Omron CX-Programmer project NewProject (CX-Programmer 9.75)

# PLC NewPLC1: CP1L M

## Global symbols (name address type ; comment)
0.00 BOOL  ; I_CYL-
0.01 BOOL  ; I_CYL+
0.02 BOOL  ; I_D-RED
0.03 BOOL  ; I_D-SILVER
0.04 BOOL  ; I_D-BLACK
0.05 BOOL  ; I_D-ENABLE V
0.06 BOOL  ; I_D-ENABLE H
0.07 BOOL  ; I_IP/FI
0.08 BOOL  ; I_PB START
0.09 BOOL  ; I_PB STOP
0.10 BOOL  ; I_SELECTOR
0.11 BOOL  ; I_RESET
100.00 BOOL  ; O_CYLINDER
100.01 BOOL  ; O_GRIPPER
100.02 BOOL  ; O_BIT 1
100.03 BOOL  ; O_BIT 2
100.04 BOOL  ; O_BIT 3
100.05 BOOL  ; O_ENABLE VERTICAL
100.06 BOOL  ; O_ENABLE HORIZONTAL
100.07 BOOL  ; O_START LAMP
101.00 BOOL  ; O_RESET LAMP
101.01 BOOL  ; O_Q1 LAMP
101.02 BOOL  ; O_Q2 LAMP
101.03 BOOL  ; O_Q4 LAMP
10.00 BOOL  ; O_IM_CYLINDER
10.01 BOOL  ; O_IM_GRIPPER
10.02 BOOL  ; O_IM_BIT 1
10.03 BOOL  ; O_IM_BIT 2
10.04 BOOL  ; O_IM_BIT 3
10.05 BOOL  ; O_IM_ENABLE VERTICAL
10.06 BOOL  ; O_IM_ENABLE HORIZONTAL
10.07 BOOL  ; O_IM_START LAMP
11.00 BOOL  ; O_IM_RESET LAMP
11.01 BOOL  ; O_IM_Q1 LAMP
11.02 BOOL  ; O_IM_Q2 LAMP
11.03 BOOL  ; O_IM_Q4 LAMP
11.04 BOOL  ; O_IM_PROGRAM BLINK
20.01 BOOL  ; SEQ1
20.02 BOOL  ; SEQ2
20.03 BOOL  ; SEQ3
20.04 BOOL  ; SEQ4
20.05 BOOL  ; SEQ5
20.06 BOOL  ; SEQ6
20.07 BOOL  ; SEQ7
20.08 BOOL  ; SEQ8
20.09 BOOL  ; SEQ9
20.10 BOOL  ; SEQ10
20.11 BOOL  ; SEQ11
20.12 BOOL  ; SEQ12
20.13 BOOL  ; SEQ13
20.14 BOOL  ; SEQ14
20.15 BOOL  ; SEQ15
21.06 BOOL  ; SEQ16
21.07 BOOL  ; SEQ17
21.08 BOOL  ; SEQ18
21.09 BOOL  ; SEQ19
22.00 BOOL  ; SEQ20
22.01 BOOL  ; SEQ21
22.02 BOOL  ; SEQ22
22.03 BOOL  ; SEQ23
30.01 BOOL  ; P_CAL1
30.02 BOOL  ; P_CAL2
30.03 BOOL  ; P_CAL3
30.04 BOOL  ; P_CAL4
30.05 BOOL  ; P_CAL5
30.06 BOOL  ; P_CAL6
30.07 BOOL  ; WP_RED
30.08 BOOL  ; WP_SILVER
30.09 BOOL  ; WP_BLACK
30.10 BOOL  ; CALIBRATION ON
30.11 BOOL  ; P_S_STOP-FUNCTION
30.12 BOOL  ; P_EMG-ACTIVE
30.13 BOOL  ; P_CAL-LAMP
30.14 BOOL  ; P_N_Send/5s
30.15 BOOL  ; P_ST_OFF LAMP
31.00 BOOL  ; P_EMERGENCY-1
31.01 BOOL  ; P_EMERGENCY-2
31.02 BOOL  ; P_EMERGENCY-3
31.03 BOOL  ; P_EMERGENCY-4
31.04 BOOL  ; DEACT WHEN RESET ON
32.00 BOOL  ; P_RST-SEQ1
32.01 BOOL  ; P_RST-SEQ2
32.02 BOOL  ; P_RST-SEQ3
32.03 BOOL  ; P_RST-SEQ4
32.04 BOOL  ; P_RST-SEQ5
32.05 BOOL  ; P_RST-SEQ6
32.06 BOOL  ; P_RST-SEQ7
32.07 BOOL  ; P_RST-SEQ8
32.08 BOOL  ; P_RST-SEQ9
32.09 BOOL  ; MANUAL RESET
32.10 BOOL  ; PB RESET HELPER
40.01 BOOL  ; SEQ-1
40.02 BOOL  ; SEQ-2
40.03 BOOL  ; SEQ-3
40.04 BOOL  ; SEQ-4
40.05 BOOL  ; SEQ-5
40.06 BOOL  ; SEQ-6
40.07 BOOL  ; SEQ-7
40.08 BOOL  ; SEQ-8
40.09 BOOL  ; SEQ-9
40.10 BOOL  ; SEQ-10
40.11 BOOL  ; SEQ-11
40.12 BOOL  ; SEQ-12
40.13 BOOL  ; SEQ-13
40.14 BOOL  ; SEQ-14
40.15 BOOL  ; SEQ-15
70.00 BOOL  ; HAPUS
70.01 BOOL  ; UBAH HMI UNTUK NON AKTIFKAN SELFHOLDING
70.02 BOOL  ; EMG PROTOTYPE
70.03 BOOL  ; TRIAL
70.04 BOOL  ; TRIAL-2
80.00 BOOL  ; CALIBRATION V
80.01 BOOL  ; LT1
80.02 BOOL  ; LT2
80.03 BOOL  ; LT3
80.04 BOOL  ; HOME
80.05 BOOL  ; PICKUP
80.07 BOOL  ; S_MOVE-V
80.08 BOOL  ; HELPER SEQ-V
80.09 BOOL  ; HELPER SEQ-V
80.10 BOOL  ; HELPER SEQ-V3
81.01 BOOL  ; POSITION 1
81.02 BOOL  ; POSITION 2
81.03 BOOL  ; POSITION 3
81.04 BOOL  ; POSITION 4
81.05 BOOL  ; POSITION 5
81.06 BOOL  ; POSITION 6
81.07 BOOL  ; HOME
81.08 BOOL  ; CALIBRATION
81.09 BOOL  ; S_MOVE-H
81.10 BOOL  ; HELPER SEQ-H
81.11 BOOL  ; HELPER SEQ-H-2
81.12 BOOL  ; HELPER SEQ-H-3
81.13 BOOL  ; HELPER H
85.00 BOOL  ; PL_LA_RED-L1
85.01 BOOL  ; PL_LA_RED-L2
85.02 BOOL  ; PL_LA_RED-L3
85.03 BOOL  ; PL_LA_SILVER-L1
85.04 BOOL  ; PL_LA_SILVER-L2
85.05 BOOL  ; PL_LA_SILVER-L3
85.06 BOOL  ; PL_LA_BLACK-L1
85.07 BOOL  ; PL_LA_BLACK-L2
85.08 BOOL  ; PL_LA_BLACK-L3
86.01 BOOL  ; PP_L3_P1
86.02 BOOL  ; PP_L3_P2
86.03 BOOL  ; PP_L3_P3
86.04 BOOL  ; PP_L3_P4
86.05 BOOL  ; PP_L3_P5
86.06 BOOL  ; PP_L3_P6
87.01 BOOL  ; PP_L2_P1
87.02 BOOL  ; PP_L2_P2
87.03 BOOL  ; PP_L2_P3
87.04 BOOL  ; PP_L2_P4
87.05 BOOL  ; PP_L2_P5
87.06 BOOL  ; PP_L2_P6
88.01 BOOL  ; PP_L1_P1
88.02 BOOL  ; PP_L1_P2
88.03 BOOL  ; PP_L1_P3
88.04 BOOL  ; PP_L1_P4
88.05 BOOL  ; PP_L1_P5
88.06 BOOL  ; PP_L1_P6
90.00 BOOL  ; TESTING_BIT1
90.01 BOOL  ; TESTING BIT 2
90.02 BOOL  ; TESTING BIT 3
90.04 BOOL  ; TESTING VERTICAL
90.05 BOOL  ; TESTING HORIZONTAL
D0 CHANNEL  ; CAL-ON
D10 CHANNEL  ; SAVE POSISI LV-1
D11 CHANNEL  ; D_BIT1
D12 CHANNEL  ; D_BIT2
D13 CHANNEL  ; D_BIT3
D14 CHANNEL  ; PL_LEVEL-TARGET
D15 CHANNEL  ; PL_LEVEL TARGET
D16 CHANNEL  ; SH_POSITION TARGET MANUAL
D17 CHANNEL  ; PP_Position Target
D18 CHANNEL  ; S_READ SEQUENCE
D19 CHANNEL  ; P_Valid Color
D2 CHANNEL  ; LEVEL 3 POS COUNT
D20 CHANNEL  ; TOTAL RED
D21 CHANNEL  ; TOTAL SILVER
D22 CHANNEL  ; TOTAL BLACK
D3 CHANNEL  ; LEVEL 2 POS COUNT
D4 CHANNEL  ; LEVEL 1 POS COUNT
D41 CHANNEL  ; P_SEQ ACTIVE
D42 CHANNEL  ; P_RST-SEQ_ACTIVE
D5 CHANNEL  ; RED LEVEL LOGIC
D6 CHANNEL  ; SILVER LEVEL LOGIC
D7 CHANNEL  ; BLACK LEVEL LOGIC
D8 CHANNEL  ; SAVE POSISI LV-3
D9 CHANNEL  ; SAVE POSISI LV-2
D91 CHANNEL  ; SEQ-H/V_SH/V_BIT1
D92 CHANNEL  ; SEQ-H/V_SH/V_BIT2
D93 CHANNEL  ; SEQ-H/V_SH/V_BIT3
D94 CHANNEL  ; SEQ-V_ON
D95 CHANNEL  ; SEQ-H_ON
D96 CHANNEL  ; SEQ-V_SEND
D97 CHANNEL  ; SEQ-H_SEND
H0.00 BOOL  ; H_M_I_CYL-
H0.01 BOOL  ; H_M_I_CYL+
H0.02 BOOL  ; H_M_I_D-RED
H0.03 BOOL  ; H_M_I_D-SILVER
H0.04 BOOL  ; H_M_I_D-BLACK
H0.05 BOOL  ; H_M_I_D-ENABLE V
H0.06 BOOL  ; H_M_I_D-ENABLE H
H0.07 BOOL  ; H_M_I_IP/FI
H0.08 BOOL  ; H_M_I_PB START
H0.09 BOOL  ; H_M_I_PB STOP
H0.10 BOOL  ; H_M_I_SELECTOR
H0.11 BOOL  ; H_M_I_RESET
H0.12 BOOL  ; H_M_O_CYLINDER
H0.13 BOOL  ; H_M_O_GRIPPER
H0.14 BOOL  ; H_M_O_BIT 1
H0.15 BOOL  ; H_M_O_BIT 2
H10.00 BOOL  ; H_M_O_CYLINDER
H10.00 BOOL  ; H_C_O_CYLINDER
H10.01 BOOL  ; H_M_O_GRIPPER
H10.01 BOOL  ; H_C_O_GRIPPER
H10.02 BOOL  ; H_M_O_BIT 1
H10.02 BOOL  ; H_C_O_BIT 1
H10.03 BOOL  ; H_M_O_BIT 2
H10.03 BOOL  ; H_C_O_BIT 2
H10.04 BOOL  ; H_M_O_BIT 3
H10.04 BOOL  ; H_C_O_BIT 3
H10.05 BOOL  ; H_M_O_ENABLE VERTICAL
H10.05 BOOL  ; H_C_O_ENABLE VERTICAL
H10.06 BOOL  ; H_M_O_ENABLE HORIZONTAL
H10.06 BOOL  ; H_C_O_ENABLE HORIZONTAL
H10.07 BOOL  ; H_M_O_START LAMP
H11.00 BOOL  ; H_M_O_RESET LAMP
H11.00 BOOL  ; H_C_O_RESET LAMP
H11.01 BOOL  ; H_M_O_Q1 LAMP
H11.01 BOOL  ; H_C_O_Q1 LAMP
H11.02 BOOL  ; H_M_O_Q2 LAMP
H11.02 BOOL  ; H_C_O_Q2 LAMP
H11.03 BOOL  ; H_M_O_Q4 LAMP
H11.03 BOOL  ; H_C_O_Q4 LAMP
H11.08 BOOL  ; H_C_I_PB START
H11.09 BOOL  ; H_C_I_PB STOP
H11.10 BOOL  ; H_C_I_SELECTOR
H11.11 BOOL  ; H_C_I_RESET
H1.00 BOOL  ; H_M_O_BIT 3
H1.01 BOOL  ; H_M_O_ENABLE VERTICAL
H1.02 BOOL  ; H_M_O_ENABLE HORIZONTAL
H1.03 BOOL  ; H_M_O_START LAMP
H1.04 BOOL  ; H_M_O_RESET LAMP
H1.05 BOOL  ; H_M_O_Q1 LAMP
H1.06 BOOL  ; H_M_O_Q2 LAMP
H1.07 BOOL  ; H_M_O_Q4 LAMP
H1.08 BOOL  ; H_P_NOTIF-3 FULL
H1.09 BOOL  ; H_P_NOTIF-2 FULL
H1.10 BOOL  ; H_P_NOTIF-1 FULL
H1.11 BOOL  ; HMI_O_IM_NOTF MANUAL ON TO HMI
H1.12 BOOL  ; H_P_STOP ON
H1.13 BOOL  ; H_P_EMERGENCY ON
H1.14 BOOL  ; H_P_RESET ON
H1.15 BOOL  ; H_P_SEQ OVERTIME
H30.00 BOOL  ; HMI_C_MANUAL PAGE
H31.00 BOOL  ; HMI_O_IM_CONNECTION CHECK
H31.01 BOOL  ; HMI_P_RESET
H31.02 BOOL  ; HMI_P_C_CALIBRATION
H35.00 BOOL  ; LEVEL 1
H35.01 BOOL  ; LEVEL 2
H35.02 BOOL  ; LEVEL 3
H40.14 BOOL  ; Helper_SVG
H40.15 BOOL  ; Pending_on nodered
H80.00 BOOL  ; HMI_CAL-V
H80.01 BOOL  ; HMI_LT1
H80.02 BOOL  ; HMI_LT2
H80.03 BOOL  ; HMI_LT3
H80.04 BOOL  ; HMI_HOME-V
H80.05 BOOL  ; HMI_PICKUP
H81.01 BOOL  ; HMI_POS1
H81.02 BOOL  ; HMI_POS2
H81.03 BOOL  ; HMI_POS3
H81.04 BOOL  ; HMI_POS4
H81.05 BOOL  ; HMI_POS5
H81.06 BOOL  ; HMI_POS6
H81.07 BOOL  ; HMI_HOME-H
H81.08 BOOL  ; HMI_CAL-H
H85.00 BOOL  ; HMI_RED_L-1
H85.01 BOOL  ; HMI_RED_L-2
H85.02 BOOL  ; HMI_RED_L-3
H85.03 BOOL  ; HMI_SILVER_L-1
H85.04 BOOL  ; HMI_SILVER_L-2
H85.05 BOOL  ; HMI_SILVER_L-3
H85.06 BOOL  ; HMI_BLACK_L-1
H85.07 BOOL  ; HMI_BLACK_L-2
H85.08 BOOL  ; HMI_BLACK_L-3
T0000 BOOL  ; Delay Detect Color
T0001 BOOL  ; DELAY GRIPPER
T0002 BOOL  ; DELAY GRIPPER
T0009 BOOL  ; T_SET
T0010 BOOL  ; T_SEND
T0021 BOOL  ; HELPER Y-
T0022 BOOL  ; DELAY GRIP
T0023 BOOL  ; DELAY CYL-
T0024 BOOL  ; HELPER CAL
T0025 BOOL  ; HELPER CAL-2
T0026 BOOL  ; HELPER CYL-
T0027 BOOL  ; P_CAL_DELAY H
T0029 BOOL  ; DELAY KE ALAMAT
T0030 BOOL  ; DELAY KE POS
T0031 BOOL  ; HELPER SEQ31
T0032 BOOL  ; HELPER SEQ 13
T0033 BOOL  ; T_HELPER RST-SEQ1
T0034 BOOL  ; T_HELPER RST-SEQ2
T0035 BOOL  ; T_HELPER RST-SEQ3
T0036 BOOL  ; T_HELPER RST-SEQ4
T0037 BOOL  ; T_HELPER RST-SEQ5
T0038 BOOL  ; T_HELPER RST-SEQ6
T0039 BOOL  ; T_HELPER RST-SEQ7
T0040 BOOL  ; T_HELPER RST-SEQ8
T0051 BOOL  ; HELPER SEQ1
T0060 BOOL  ; T_CAL SET
T0061 BOOL  ; T_CAL SEND
T0064 BOOL  ; tes
T0065 BOOL  ; tes
T0090 BOOL  ; T SEND
T0091 BOOL  ; RESET
T0092 BOOL  ; TIMER SET HORIZONTAL
T0093 BOOL  ; RESET
T0095 BOOL  ; HELPER SEQ
T0096 BOOL  ; T_HELPER_SH

## Program NewProgram1 (cyclic task 0)
Local symbols
p_On BOOL

### Section PROGRAM

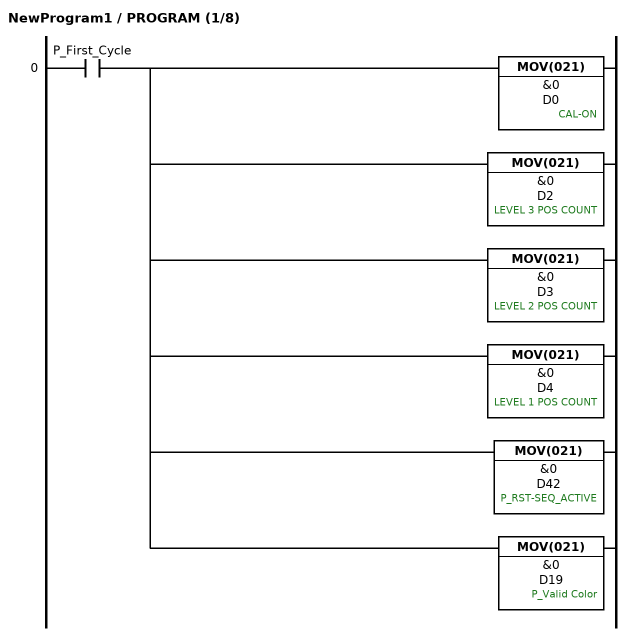
; rung 0
LD P_First_Cycle
MOV(021) &0 D0  ; CAL-ON
MOV(021) &0 D2  ; LEVEL 3 POS COUNT
MOV(021) &0 D3  ; LEVEL 2 POS COUNT
MOV(021) &0 D4  ; LEVEL 1 POS COUNT
MOV(021) &0 D42  ; P_RST-SEQ_ACTIVE
MOV(021) &0 D19  ; P_Valid Color

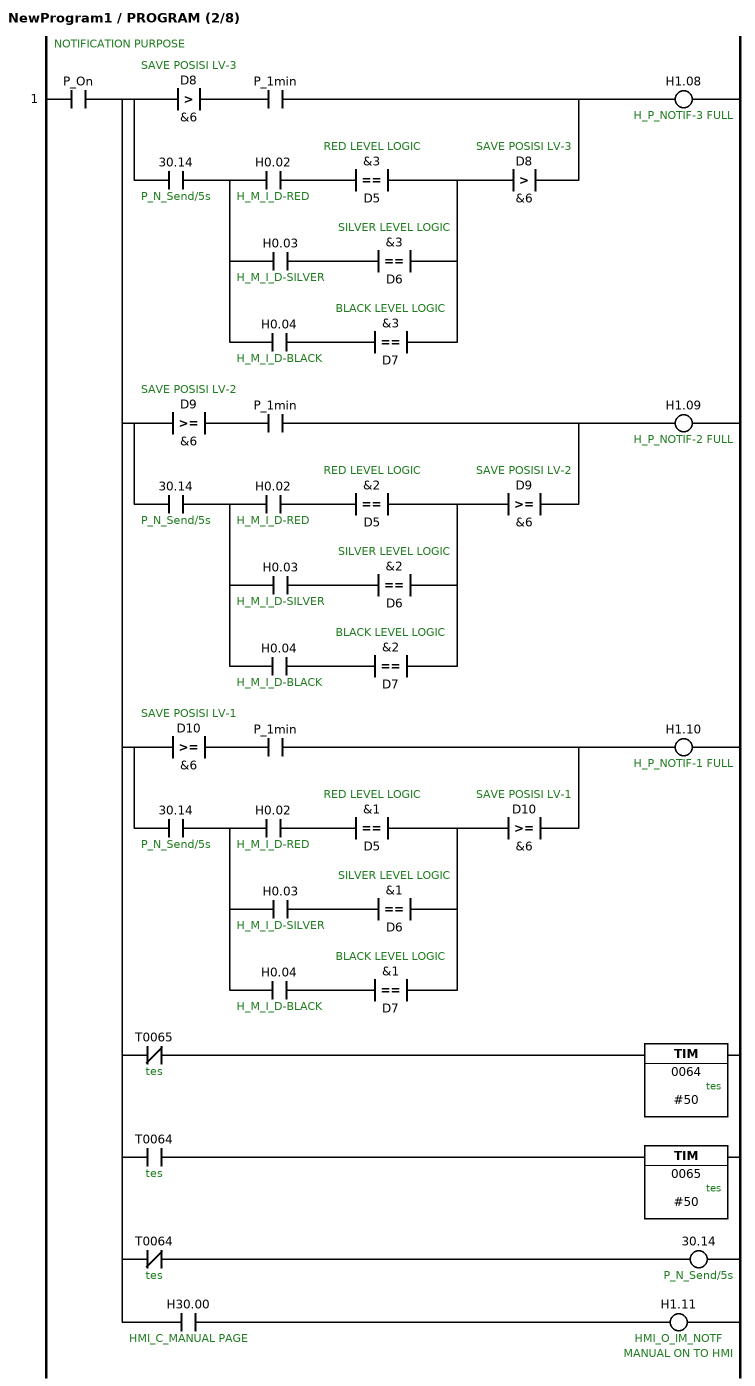
; rung 1: NOTIFICATION PURPOSE
LD P_On
OUT TR0
LD>(320) D8 &6  ; SAVE POSISI LV-3
AND P_1min
LD 30.14  ; P_N_Send/5s
LD H0.02  ; H_M_I_D-RED
AND=(300) &3 D5  ; RED LEVEL LOGIC
LD H0.03  ; H_M_I_D-SILVER
AND=(300) &3 D6  ; SILVER LEVEL LOGIC
ORLD
LD H0.04  ; H_M_I_D-BLACK
AND=(300) &3 D7  ; BLACK LEVEL LOGIC
ORLD
ANDLD
AND>(320) D8 &6  ; SAVE POSISI LV-3
ORLD
ANDLD
OUT H1.08  ; H_P_NOTIF-3 FULL
LD TR0
LD>=(325) D9 &6  ; SAVE POSISI LV-2
AND P_1min
LD 30.14  ; P_N_Send/5s
LD H0.02  ; H_M_I_D-RED
AND=(300) &2 D5  ; RED LEVEL LOGIC
LD H0.03  ; H_M_I_D-SILVER
AND=(300) &2 D6  ; SILVER LEVEL LOGIC
ORLD
LD H0.04  ; H_M_I_D-BLACK
AND=(300) &2 D7  ; BLACK LEVEL LOGIC
ORLD
ANDLD
AND>=(325) D9 &6  ; SAVE POSISI LV-2
ORLD
ANDLD
OUT H1.09  ; H_P_NOTIF-2 FULL
LD TR0
LD>=(325) D10 &6  ; SAVE POSISI LV-1
AND P_1min
LD 30.14  ; P_N_Send/5s
LD H0.02  ; H_M_I_D-RED
AND=(300) &1 D5  ; RED LEVEL LOGIC
LD H0.03  ; H_M_I_D-SILVER
AND=(300) &1 D6  ; SILVER LEVEL LOGIC
ORLD
LD H0.04  ; H_M_I_D-BLACK
AND=(300) &1 D7  ; BLACK LEVEL LOGIC
ORLD
ANDLD
AND>=(325) D10 &6  ; SAVE POSISI LV-1
ORLD
ANDLD
OUT H1.10  ; H_P_NOTIF-1 FULL
LD TR0
ANDNOT T0065  ; tes
TIM 0064 #50  ; tes
LD TR0
AND T0064  ; tes
TIM 0065 #50  ; tes
LD TR0
ANDNOT T0064  ; tes
OUT 30.14  ; P_N_Send/5s
LD TR0
AND H30.00  ; HMI_C_MANUAL PAGE
OUT H1.11  ; HMI_O_IM_NOTF MANUAL ON TO HMI

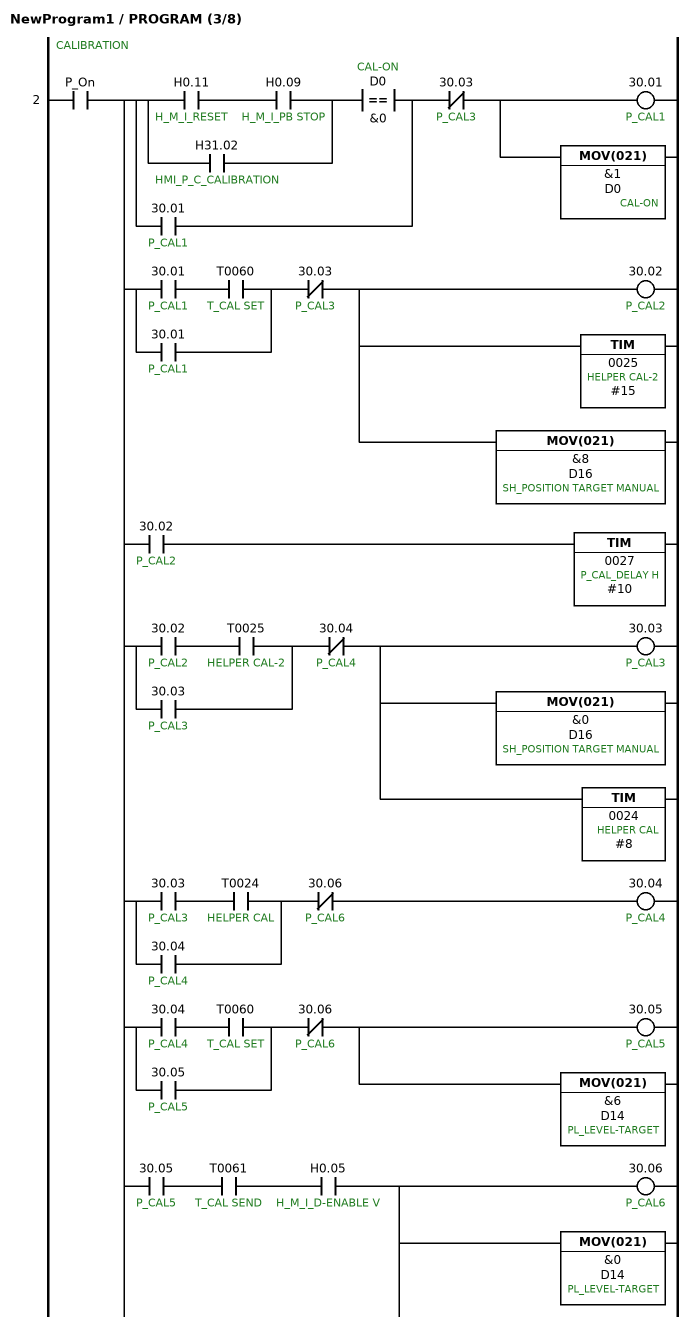

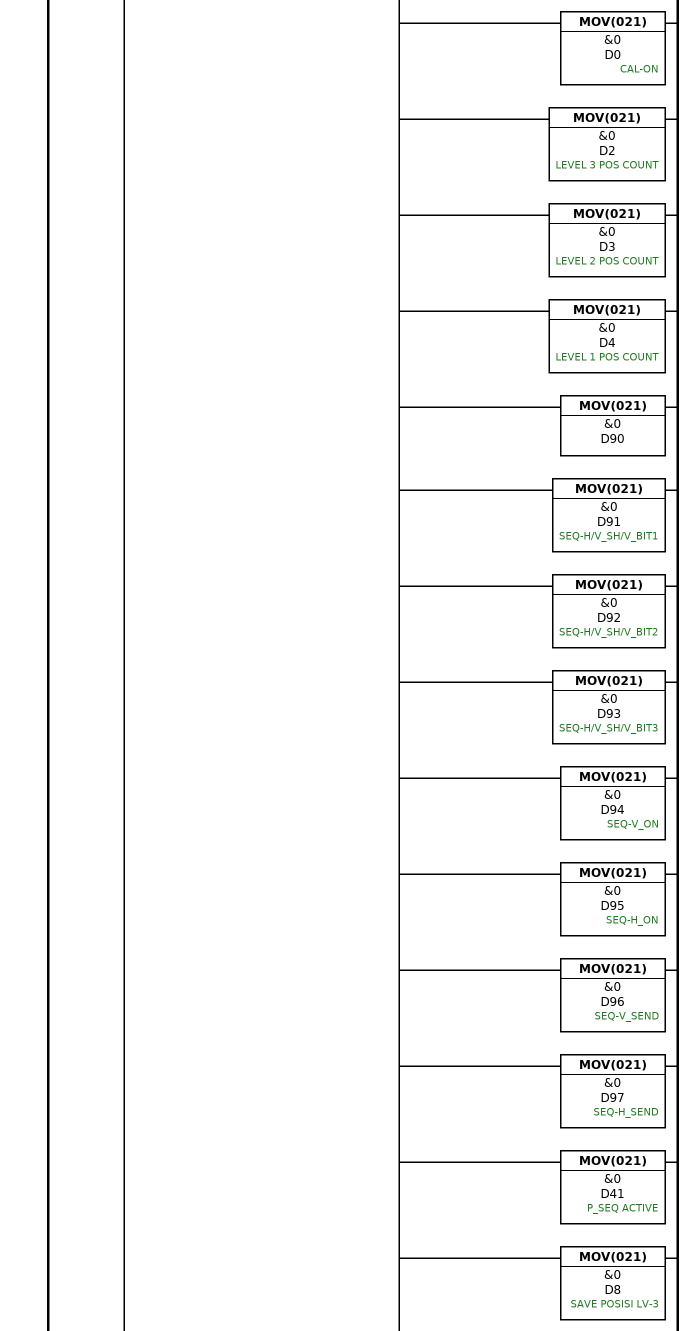

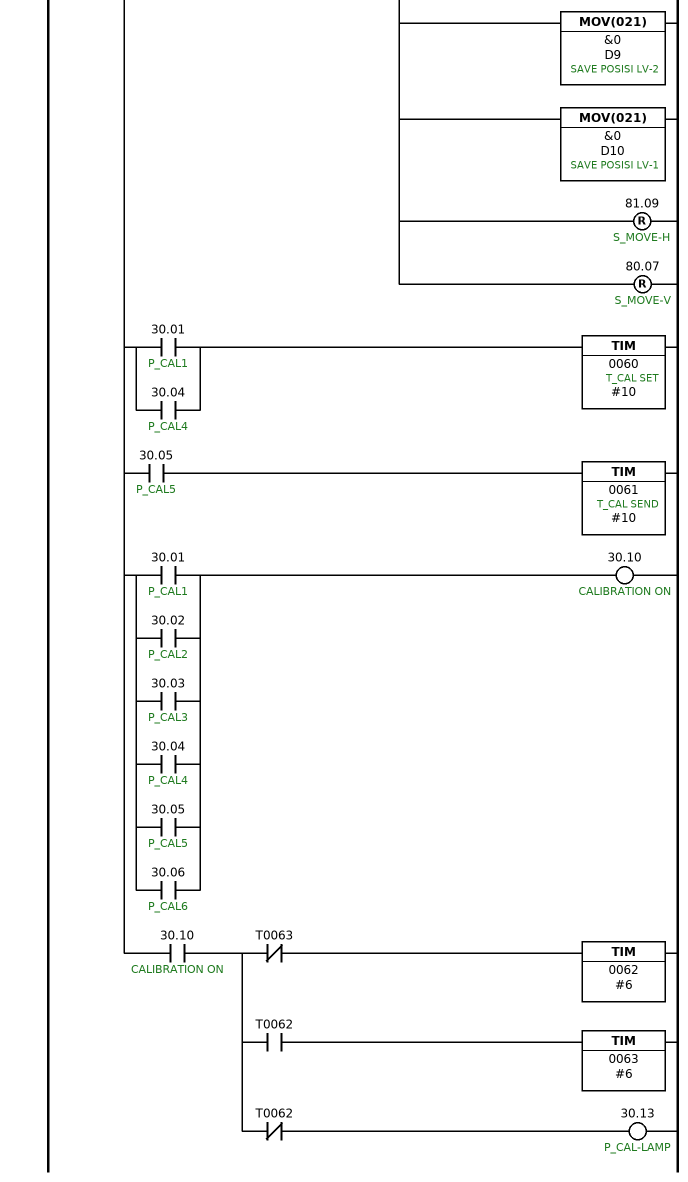
; rung 2: CALIBRATION
LD P_On
OUT TR0
LD H0.11  ; H_M_I_RESET
AND H0.09  ; H_M_I_PB STOP
OR H31.02  ; HMI_P_C_CALIBRATION
AND=(300) D0 &0  ; CAL-ON
OR 30.01  ; P_CAL1
ANDLD
ANDNOT 30.03  ; P_CAL3
OUT 30.01  ; P_CAL1
MOV(021) &1 D0  ; CAL-ON
LD TR0
LD 30.01  ; P_CAL1
AND T0060  ; T_CAL SET
OR 30.01  ; P_CAL1
ANDLD
ANDNOT 30.03  ; P_CAL3
OUT 30.02  ; P_CAL2
TIM 0025 #15  ; HELPER CAL-2
MOV(021) &8 D16  ; SH_POSITION TARGET MANUAL
LD TR0
AND 30.02  ; P_CAL2
TIM 0027 #10  ; P_CAL_DELAY H
LD TR0
LD 30.02  ; P_CAL2
AND T0025  ; HELPER CAL-2
OR 30.03  ; P_CAL3
ANDLD
ANDNOT 30.04  ; P_CAL4
OUT 30.03  ; P_CAL3
MOV(021) &0 D16  ; SH_POSITION TARGET MANUAL
TIM 0024 #8  ; HELPER CAL
LD TR0
LD 30.03  ; P_CAL3
AND T0024  ; HELPER CAL
OR 30.04  ; P_CAL4
ANDLD
ANDNOT 30.06  ; P_CAL6
OUT 30.04  ; P_CAL4
LD TR0
LD 30.04  ; P_CAL4
AND T0060  ; T_CAL SET
OR 30.05  ; P_CAL5
ANDLD
ANDNOT 30.06  ; P_CAL6
OUT 30.05  ; P_CAL5
MOV(021) &6 D14  ; PL_LEVEL-TARGET
LD TR0
AND 30.05  ; P_CAL5
AND T0061  ; T_CAL SEND
AND H0.05  ; H_M_I_D-ENABLE V
OUT 30.06  ; P_CAL6
MOV(021) &0 D14  ; PL_LEVEL-TARGET
MOV(021) &0 D0  ; CAL-ON
MOV(021) &0 D2  ; LEVEL 3 POS COUNT
MOV(021) &0 D3  ; LEVEL 2 POS COUNT
MOV(021) &0 D4  ; LEVEL 1 POS COUNT
MOV(021) &0 D90
MOV(021) &0 D91  ; SEQ-H/V_SH/V_BIT1
MOV(021) &0 D92  ; SEQ-H/V_SH/V_BIT2
MOV(021) &0 D93  ; SEQ-H/V_SH/V_BIT3
MOV(021) &0 D94  ; SEQ-V_ON
MOV(021) &0 D95  ; SEQ-H_ON
MOV(021) &0 D96  ; SEQ-V_SEND
MOV(021) &0 D97  ; SEQ-H_SEND
MOV(021) &0 D41  ; P_SEQ ACTIVE
MOV(021) &0 D8  ; SAVE POSISI LV-3
MOV(021) &0 D9  ; SAVE POSISI LV-2
MOV(021) &0 D10  ; SAVE POSISI LV-1
RSET 81.09  ; S_MOVE-H
RSET 80.07  ; S_MOVE-V
LD TR0
LD 30.01  ; P_CAL1
OR 30.04  ; P_CAL4
ANDLD
TIM 0060 #10  ; T_CAL SET
LD TR0
AND 30.05  ; P_CAL5
TIM 0061 #10  ; T_CAL SEND
LD TR0
LD 30.01  ; P_CAL1
OR 30.02  ; P_CAL2
OR 30.03  ; P_CAL3
OR 30.04  ; P_CAL4
OR 30.05  ; P_CAL5
OR 30.06  ; P_CAL6
ANDLD
OUT 30.10  ; CALIBRATION ON
LD TR0
AND 30.10  ; CALIBRATION ON
OUT TR0
ANDNOT T0063
TIM 0062 #6
LD TR0
AND T0062
TIM 0063 #6
LD TR0
ANDNOT T0062
OUT 30.13  ; P_CAL-LAMP

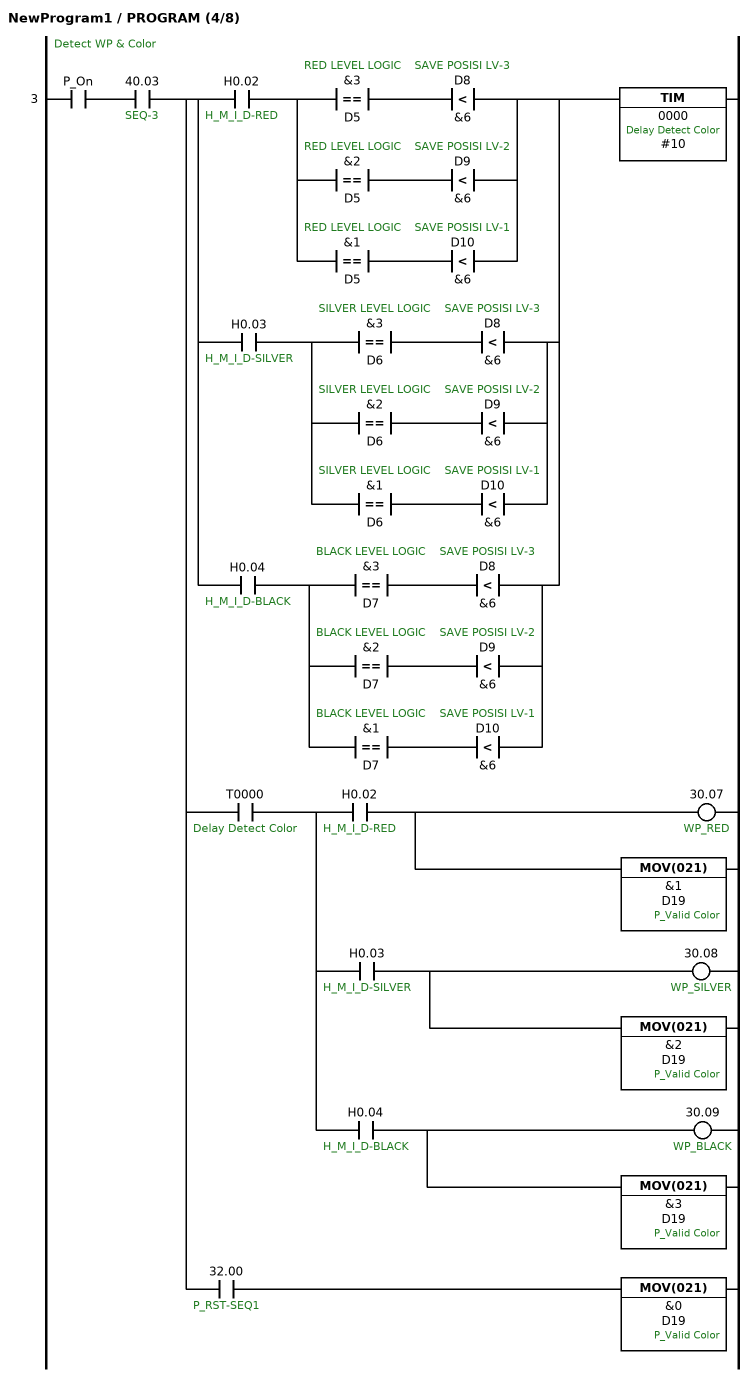
; rung 3: Detect WP & Color
LD P_On
AND 40.03  ; SEQ-3
OUT TR0
LD H0.02  ; H_M_I_D-RED
LD=(300) &3 D5  ; RED LEVEL LOGIC
AND<(310) D8 &6  ; SAVE POSISI LV-3
LD=(300) &2 D5  ; RED LEVEL LOGIC
AND<(310) D9 &6  ; SAVE POSISI LV-2
ORLD
LD=(300) &1 D5  ; RED LEVEL LOGIC
AND<(310) D10 &6  ; SAVE POSISI LV-1
ORLD
ANDLD
LD H0.03  ; H_M_I_D-SILVER
LD=(300) &3 D6  ; SILVER LEVEL LOGIC
AND<(310) D8 &6  ; SAVE POSISI LV-3
LD=(300) &2 D6  ; SILVER LEVEL LOGIC
AND<(310) D9 &6  ; SAVE POSISI LV-2
ORLD
LD=(300) &1 D6  ; SILVER LEVEL LOGIC
AND<(310) D10 &6  ; SAVE POSISI LV-1
ORLD
ANDLD
ORLD
LD H0.04  ; H_M_I_D-BLACK
LD=(300) &3 D7  ; BLACK LEVEL LOGIC
AND<(310) D8 &6  ; SAVE POSISI LV-3
LD=(300) &2 D7  ; BLACK LEVEL LOGIC
AND<(310) D9 &6  ; SAVE POSISI LV-2
ORLD
LD=(300) &1 D7  ; BLACK LEVEL LOGIC
AND<(310) D10 &6  ; SAVE POSISI LV-1
ORLD
ANDLD
ORLD
ANDLD
TIM 0000 #10  ; Delay Detect Color
LD TR0
AND T0000  ; Delay Detect Color
OUT TR1
AND H0.02  ; H_M_I_D-RED
OUT 30.07  ; WP_RED
MOV(021) &1 D19  ; P_Valid Color
LD TR1
AND H0.03  ; H_M_I_D-SILVER
OUT 30.08  ; WP_SILVER
MOV(021) &2 D19  ; P_Valid Color
LD TR1
AND H0.04  ; H_M_I_D-BLACK
OUT 30.09  ; WP_BLACK
MOV(021) &3 D19  ; P_Valid Color
LD TR0
AND 32.00  ; P_RST-SEQ1
MOV(021) &0 D19  ; P_Valid Color

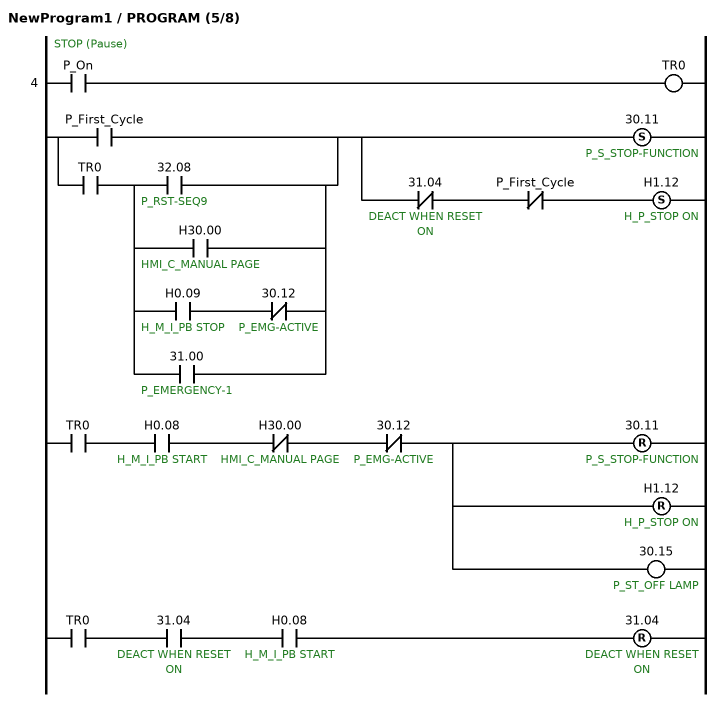
; rung 4: STOP (Pause)
LD P_First_Cycle
LD P_On
OUT TR0
LD 32.08  ; P_RST-SEQ9
OR H30.00  ; HMI_C_MANUAL PAGE
LD H0.09  ; H_M_I_PB STOP
ANDNOT 30.12  ; P_EMG-ACTIVE
ORLD
OR 31.00  ; P_EMERGENCY-1
ANDLD
ORLD
SET 30.11  ; P_S_STOP-FUNCTION
ANDNOT 31.04  ; DEACT WHEN RESET ON
ANDNOT P_First_Cycle
SET H1.12  ; H_P_STOP ON
LD TR0
AND H0.08  ; H_M_I_PB START
ANDNOT H30.00  ; HMI_C_MANUAL PAGE
ANDNOT 30.12  ; P_EMG-ACTIVE
RSET 30.11  ; P_S_STOP-FUNCTION
RSET H1.12  ; H_P_STOP ON
OUT 30.15  ; P_ST_OFF LAMP
LD TR0
AND 31.04  ; DEACT WHEN RESET ON
AND H0.08  ; H_M_I_PB START
RSET 31.04  ; DEACT WHEN RESET ON

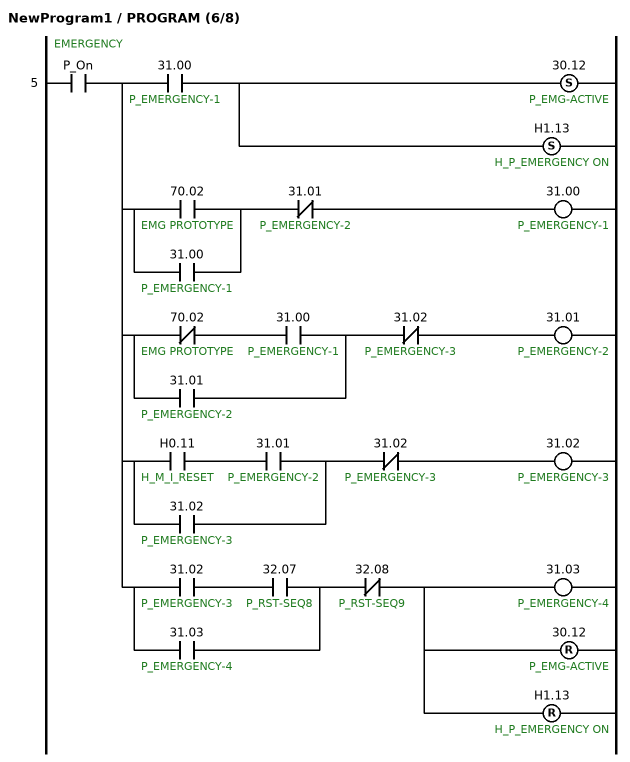
; rung 5: EMERGENCY
LD P_On
OUT TR0
AND 31.00  ; P_EMERGENCY-1
SET 30.12  ; P_EMG-ACTIVE
SET H1.13  ; H_P_EMERGENCY ON
LD TR0
LD 70.02  ; EMG PROTOTYPE
OR 31.00  ; P_EMERGENCY-1
ANDLD
ANDNOT 31.01  ; P_EMERGENCY-2
OUT 31.00  ; P_EMERGENCY-1
LD TR0
LDNOT 70.02  ; EMG PROTOTYPE
AND 31.00  ; P_EMERGENCY-1
OR 31.01  ; P_EMERGENCY-2
ANDLD
ANDNOT 31.02  ; P_EMERGENCY-3
OUT 31.01  ; P_EMERGENCY-2
LD TR0
LD H0.11  ; H_M_I_RESET
AND 31.01  ; P_EMERGENCY-2
OR 31.02  ; P_EMERGENCY-3
ANDLD
ANDNOT 31.02  ; P_EMERGENCY-3
OUT 31.02  ; P_EMERGENCY-3
LD TR0
LD 31.02  ; P_EMERGENCY-3
AND 32.07  ; P_RST-SEQ8
OR 31.03  ; P_EMERGENCY-4
ANDLD
ANDNOT 32.08  ; P_RST-SEQ9
OUT 31.03  ; P_EMERGENCY-4
RSET 30.12  ; P_EMG-ACTIVE
RSET H1.13  ; H_P_EMERGENCY ON

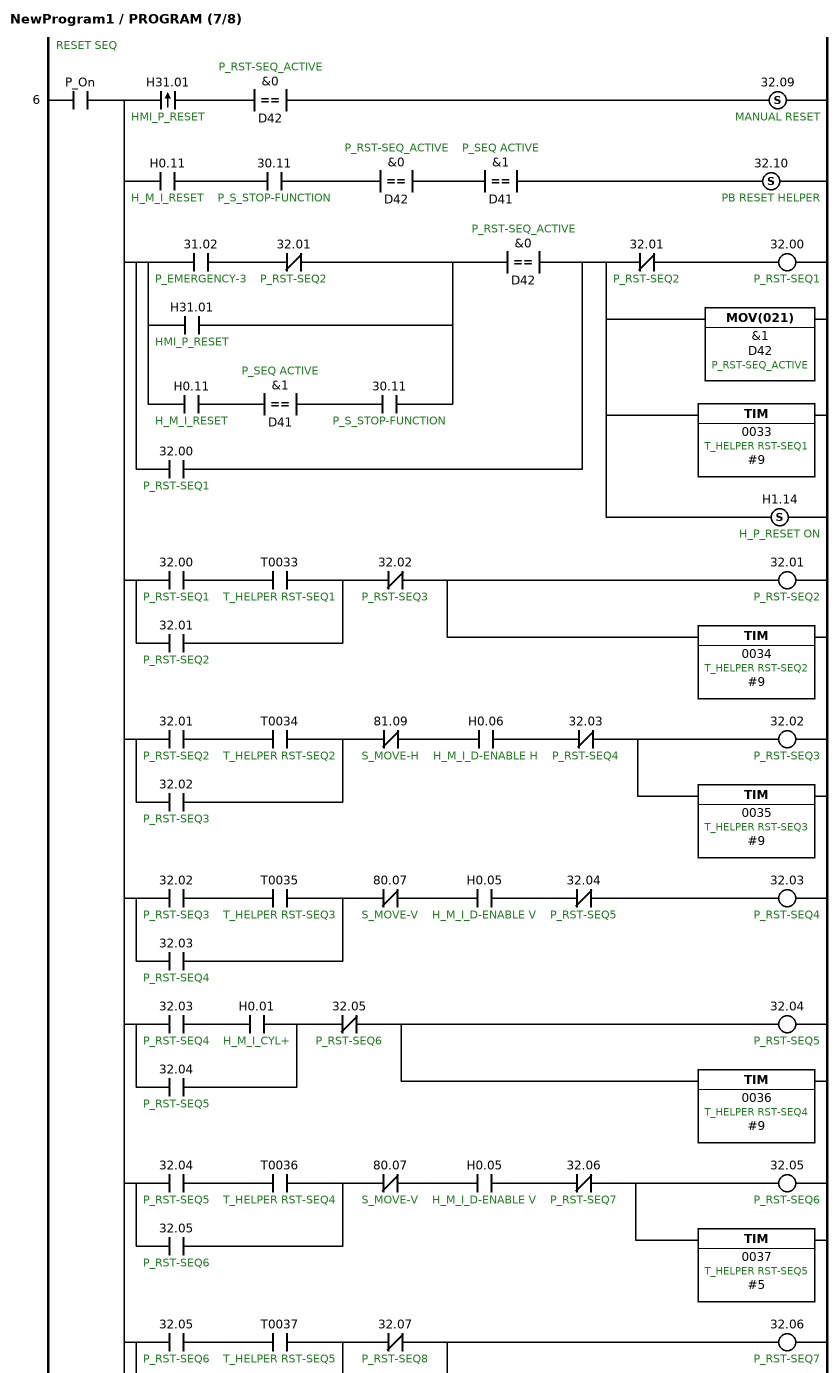

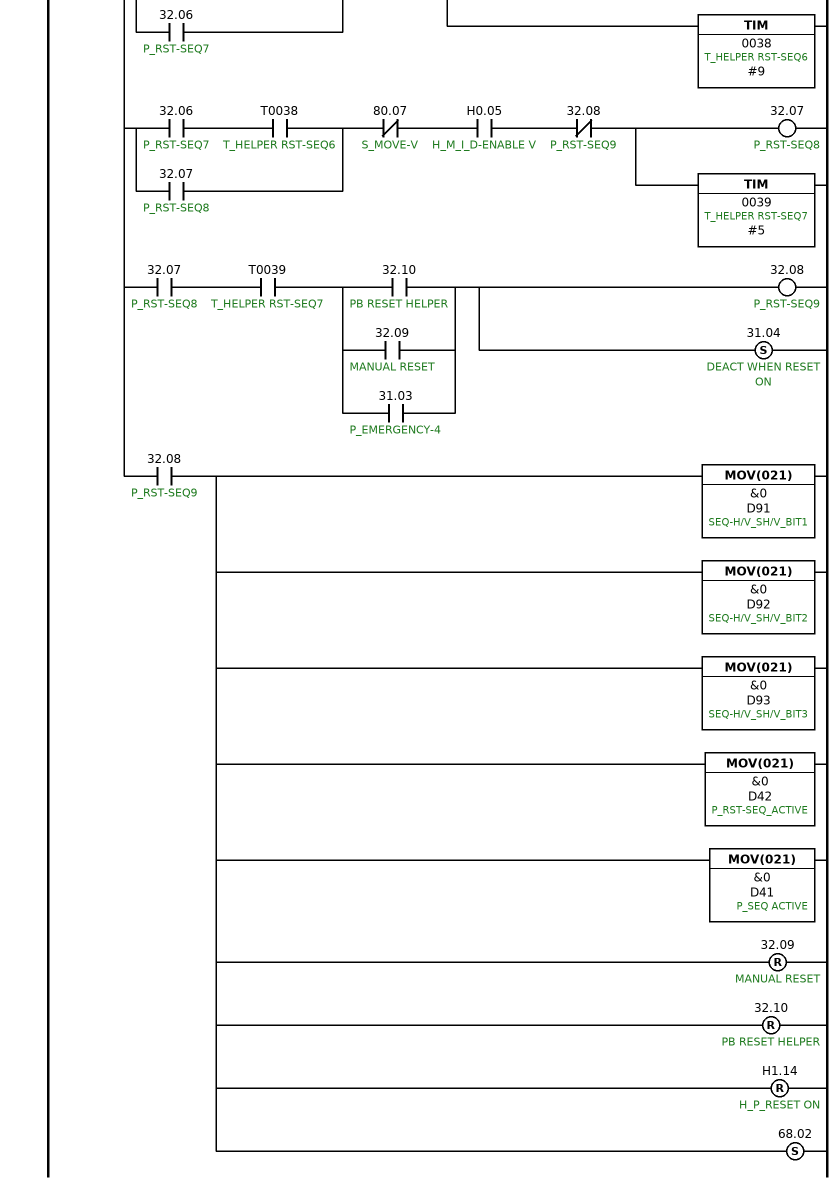
; rung 6: RESET SEQ
LD P_On
OUT TR0
@AND H31.01  ; HMI_P_RESET
AND=(300) &0 D42  ; P_RST-SEQ_ACTIVE
SET 32.09  ; MANUAL RESET
LD TR0
AND H0.11  ; H_M_I_RESET
AND 30.11  ; P_S_STOP-FUNCTION
AND=(300) &0 D42  ; P_RST-SEQ_ACTIVE
AND=(300) &1 D41  ; P_SEQ ACTIVE
SET 32.10  ; PB RESET HELPER
LD TR0
LD 31.02  ; P_EMERGENCY-3
ANDNOT 32.01  ; P_RST-SEQ2
OR H31.01  ; HMI_P_RESET
LD H0.11  ; H_M_I_RESET
AND=(300) &1 D41  ; P_SEQ ACTIVE
AND 30.11  ; P_S_STOP-FUNCTION
ORLD
AND=(300) &0 D42  ; P_RST-SEQ_ACTIVE
OR 32.00  ; P_RST-SEQ1
ANDLD
OUT TR1
ANDNOT 32.01  ; P_RST-SEQ2
OUT 32.00  ; P_RST-SEQ1
LD TR1
MOV(021) &1 D42  ; P_RST-SEQ_ACTIVE
TIM 0033 #9  ; T_HELPER RST-SEQ1
SET H1.14  ; H_P_RESET ON
LD TR0
LD 32.00  ; P_RST-SEQ1
AND T0033  ; T_HELPER RST-SEQ1
OR 32.01  ; P_RST-SEQ2
ANDLD
ANDNOT 32.02  ; P_RST-SEQ3
OUT 32.01  ; P_RST-SEQ2
TIM 0034 #9  ; T_HELPER RST-SEQ2
LD TR0
LD 32.01  ; P_RST-SEQ2
AND T0034  ; T_HELPER RST-SEQ2
OR 32.02  ; P_RST-SEQ3
ANDLD
ANDNOT 81.09  ; S_MOVE-H
AND H0.06  ; H_M_I_D-ENABLE H
ANDNOT 32.03  ; P_RST-SEQ4
OUT 32.02  ; P_RST-SEQ3
TIM 0035 #9  ; T_HELPER RST-SEQ3
LD TR0
LD 32.02  ; P_RST-SEQ3
AND T0035  ; T_HELPER RST-SEQ3
OR 32.03  ; P_RST-SEQ4
ANDLD
ANDNOT 80.07  ; S_MOVE-V
AND H0.05  ; H_M_I_D-ENABLE V
ANDNOT 32.04  ; P_RST-SEQ5
OUT 32.03  ; P_RST-SEQ4
LD TR0
LD 32.03  ; P_RST-SEQ4
AND H0.01  ; H_M_I_CYL+
OR 32.04  ; P_RST-SEQ5
ANDLD
ANDNOT 32.05  ; P_RST-SEQ6
OUT 32.04  ; P_RST-SEQ5
TIM 0036 #9  ; T_HELPER RST-SEQ4
LD TR0
LD 32.04  ; P_RST-SEQ5
AND T0036  ; T_HELPER RST-SEQ4
OR 32.05  ; P_RST-SEQ6
ANDLD
ANDNOT 80.07  ; S_MOVE-V
AND H0.05  ; H_M_I_D-ENABLE V
ANDNOT 32.06  ; P_RST-SEQ7
OUT 32.05  ; P_RST-SEQ6
TIM 0037 #5  ; T_HELPER RST-SEQ5
LD TR0
LD 32.05  ; P_RST-SEQ6
AND T0037  ; T_HELPER RST-SEQ5
OR 32.06  ; P_RST-SEQ7
ANDLD
ANDNOT 32.07  ; P_RST-SEQ8
OUT 32.06  ; P_RST-SEQ7
TIM 0038 #9  ; T_HELPER RST-SEQ6
LD TR0
LD 32.06  ; P_RST-SEQ7
AND T0038  ; T_HELPER RST-SEQ6
OR 32.07  ; P_RST-SEQ8
ANDLD
ANDNOT 80.07  ; S_MOVE-V
AND H0.05  ; H_M_I_D-ENABLE V
ANDNOT 32.08  ; P_RST-SEQ9
OUT 32.07  ; P_RST-SEQ8
TIM 0039 #5  ; T_HELPER RST-SEQ7
LD TR0
AND 32.07  ; P_RST-SEQ8
AND T0039  ; T_HELPER RST-SEQ7
LD 32.10  ; PB RESET HELPER
OR 32.09  ; MANUAL RESET
OR 31.03  ; P_EMERGENCY-4
ANDLD
OUT 32.08  ; P_RST-SEQ9
SET 31.04  ; DEACT WHEN RESET ON
LD TR0
AND 32.08  ; P_RST-SEQ9
MOV(021) &0 D91  ; SEQ-H/V_SH/V_BIT1
MOV(021) &0 D92  ; SEQ-H/V_SH/V_BIT2
MOV(021) &0 D93  ; SEQ-H/V_SH/V_BIT3
MOV(021) &0 D42  ; P_RST-SEQ_ACTIVE
MOV(021) &0 D41  ; P_SEQ ACTIVE
RSET 32.09  ; MANUAL RESET
RSET 32.10  ; PB RESET HELPER
RSET H1.14  ; H_P_RESET ON
SET 68.02

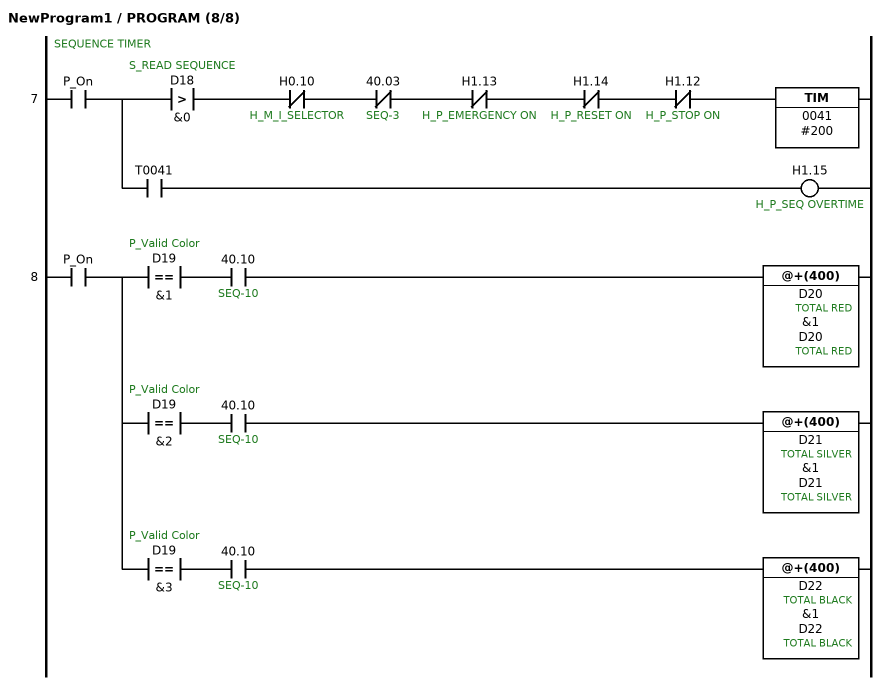
; rung 7: SEQUENCE TIMER
LD P_On
OUT TR0
AND>(320) D18 &0  ; S_READ SEQUENCE
ANDNOT H0.10  ; H_M_I_SELECTOR
ANDNOT 40.03  ; SEQ-3
ANDNOT H1.13  ; H_P_EMERGENCY ON
ANDNOT H1.14  ; H_P_RESET ON
ANDNOT H1.12  ; H_P_STOP ON
TIM 0041 #200
LD TR0
AND T0041
OUT H1.15  ; H_P_SEQ OVERTIME
; rung 8
LD P_On
OUT TR0
AND=(300) D19 &1  ; P_Valid Color
AND 40.10  ; SEQ-10
@+(400) D20 &1 D20  ; TOTAL RED
LD TR0
AND=(300) D19 &2  ; P_Valid Color
AND 40.10  ; SEQ-10
@+(400) D21 &1 D21  ; TOTAL SILVER
LD TR0
AND=(300) D19 &3  ; P_Valid Color
AND 40.10  ; SEQ-10
@+(400) D22 &1 D22  ; TOTAL BLACK

### Section PROGRAM_LEVEL

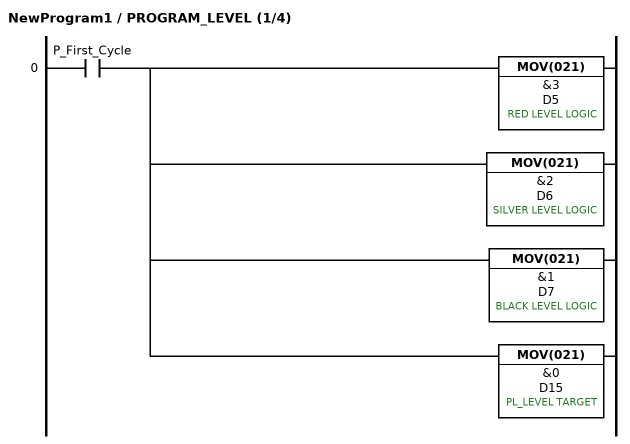
; rung 0
LD P_First_Cycle
MOV(021) &3 D5  ; RED LEVEL LOGIC
MOV(021) &2 D6  ; SILVER LEVEL LOGIC
MOV(021) &1 D7  ; BLACK LEVEL LOGIC
MOV(021) &0 D15  ; PL_LEVEL TARGET

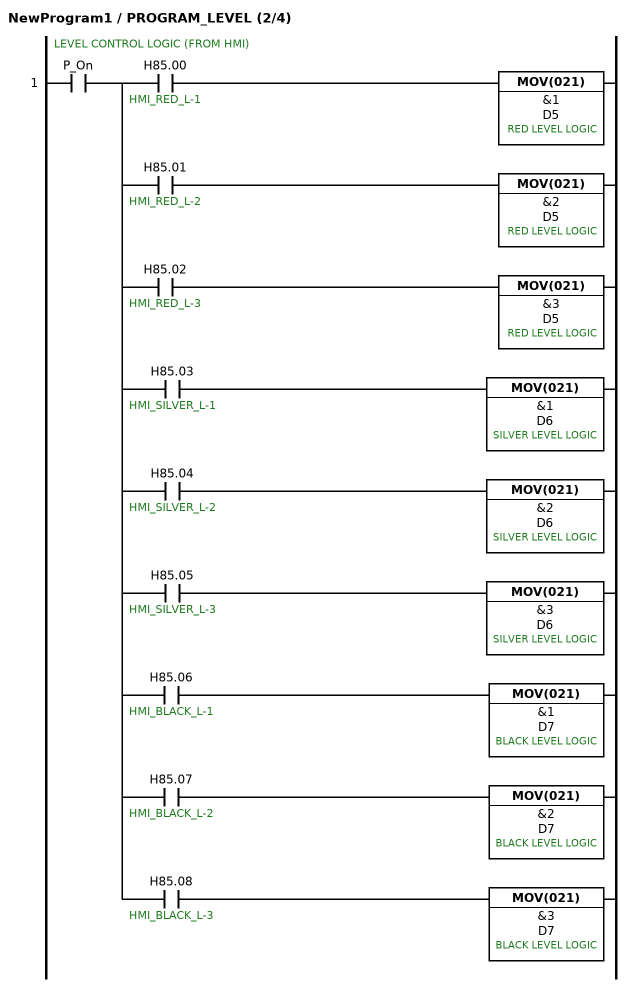
; rung 1: LEVEL CONTROL LOGIC (FROM HMI)
LD P_On
OUT TR0
AND H85.00  ; HMI_RED_L-1
MOV(021) &1 D5  ; RED LEVEL LOGIC
LD TR0
AND H85.01  ; HMI_RED_L-2
MOV(021) &2 D5  ; RED LEVEL LOGIC
LD TR0
AND H85.02  ; HMI_RED_L-3
MOV(021) &3 D5  ; RED LEVEL LOGIC
LD TR0
AND H85.03  ; HMI_SILVER_L-1
MOV(021) &1 D6  ; SILVER LEVEL LOGIC
LD TR0
AND H85.04  ; HMI_SILVER_L-2
MOV(021) &2 D6  ; SILVER LEVEL LOGIC
LD TR0
AND H85.05  ; HMI_SILVER_L-3
MOV(021) &3 D6  ; SILVER LEVEL LOGIC
LD TR0
AND H85.06  ; HMI_BLACK_L-1
MOV(021) &1 D7  ; BLACK LEVEL LOGIC
LD TR0
AND H85.07  ; HMI_BLACK_L-2
MOV(021) &2 D7  ; BLACK LEVEL LOGIC
LD TR0
AND H85.08  ; HMI_BLACK_L-3
MOV(021) &3 D7  ; BLACK LEVEL LOGIC

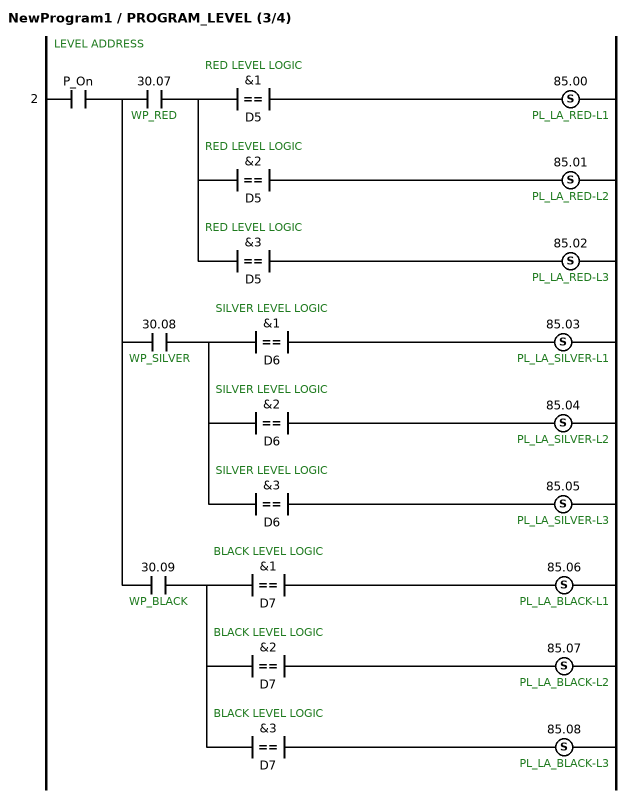
; rung 2: LEVEL ADDRESS
LD P_On
OUT TR0
AND 30.07  ; WP_RED
OUT TR1
AND=(300) &1 D5  ; RED LEVEL LOGIC
SET 85.00  ; PL_LA_RED-L1
LD TR1
AND=(300) &2 D5  ; RED LEVEL LOGIC
SET 85.01  ; PL_LA_RED-L2
LD TR1
AND=(300) &3 D5  ; RED LEVEL LOGIC
SET 85.02  ; PL_LA_RED-L3
LD TR0
AND 30.08  ; WP_SILVER
OUT TR1
AND=(300) &1 D6  ; SILVER LEVEL LOGIC
SET 85.03  ; PL_LA_SILVER-L1
LD TR1
AND=(300) &2 D6  ; SILVER LEVEL LOGIC
SET 85.04  ; PL_LA_SILVER-L2
LD TR1
AND=(300) &3 D6  ; SILVER LEVEL LOGIC
SET 85.05  ; PL_LA_SILVER-L3
LD TR0
AND 30.09  ; WP_BLACK
OUT TR0
AND=(300) &1 D7  ; BLACK LEVEL LOGIC
SET 85.06  ; PL_LA_BLACK-L1
LD TR0
AND=(300) &2 D7  ; BLACK LEVEL LOGIC
SET 85.07  ; PL_LA_BLACK-L2
LD TR0
AND=(300) &3 D7  ; BLACK LEVEL LOGIC
SET 85.08  ; PL_LA_BLACK-L3

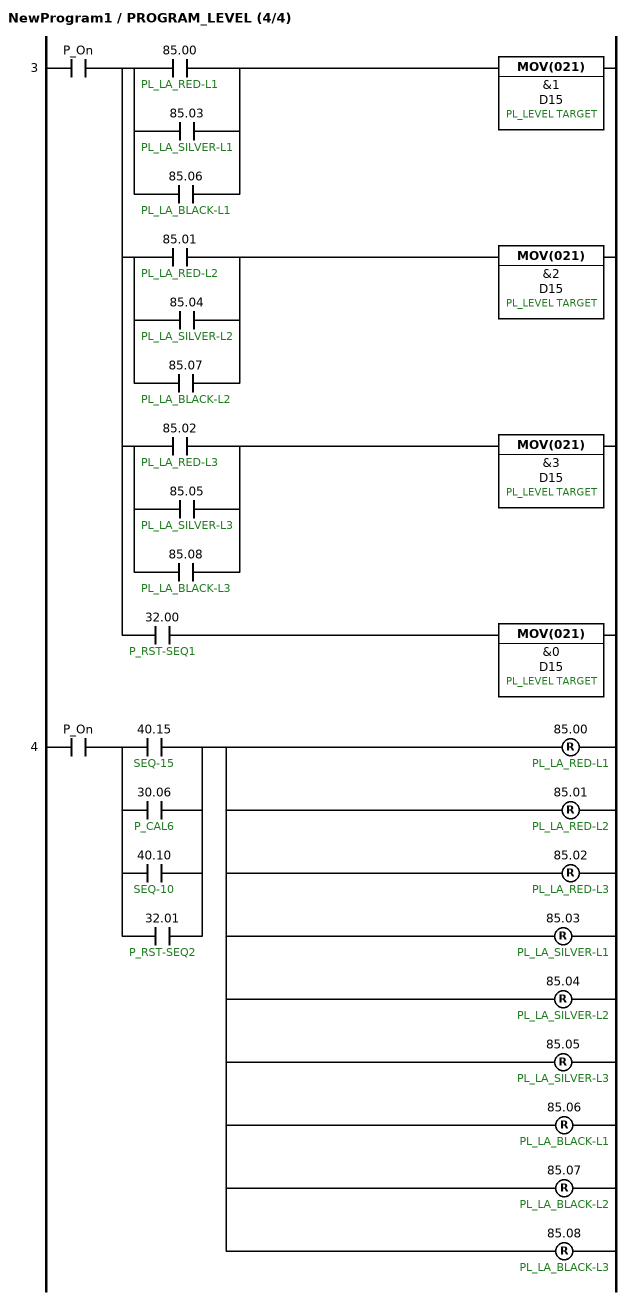
; rung 3
LD P_On
OUT TR0
LD 85.00  ; PL_LA_RED-L1
OR 85.03  ; PL_LA_SILVER-L1
OR 85.06  ; PL_LA_BLACK-L1
ANDLD
MOV(021) &1 D15  ; PL_LEVEL TARGET
LD TR0
LD 85.01  ; PL_LA_RED-L2
OR 85.04  ; PL_LA_SILVER-L2
OR 85.07  ; PL_LA_BLACK-L2
ANDLD
MOV(021) &2 D15  ; PL_LEVEL TARGET
LD TR0
LD 85.02  ; PL_LA_RED-L3
OR 85.05  ; PL_LA_SILVER-L3
OR 85.08  ; PL_LA_BLACK-L3
ANDLD
MOV(021) &3 D15  ; PL_LEVEL TARGET
LD TR0
AND 32.00  ; P_RST-SEQ1
MOV(021) &0 D15  ; PL_LEVEL TARGET
; rung 4
LD P_On
LD 40.15  ; SEQ-15
OR 30.06  ; P_CAL6
OR 40.10  ; SEQ-10
OR 32.01  ; P_RST-SEQ2
ANDLD
RSET 85.00  ; PL_LA_RED-L1
RSET 85.01  ; PL_LA_RED-L2
RSET 85.02  ; PL_LA_RED-L3
RSET 85.03  ; PL_LA_SILVER-L1
RSET 85.04  ; PL_LA_SILVER-L2
RSET 85.05  ; PL_LA_SILVER-L3
RSET 85.06  ; PL_LA_BLACK-L1
RSET 85.07  ; PL_LA_BLACK-L2
RSET 85.08  ; PL_LA_BLACK-L3

### Section PROGRAM_POSITION

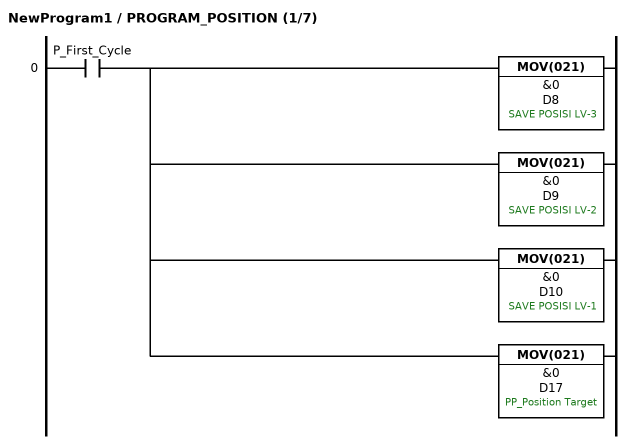
; rung 0
LD P_First_Cycle
MOV(021) &0 D8  ; SAVE POSISI LV-3
MOV(021) &0 D9  ; SAVE POSISI LV-2
MOV(021) &0 D10  ; SAVE POSISI LV-1
MOV(021) &0 D17  ; PP_Position Target

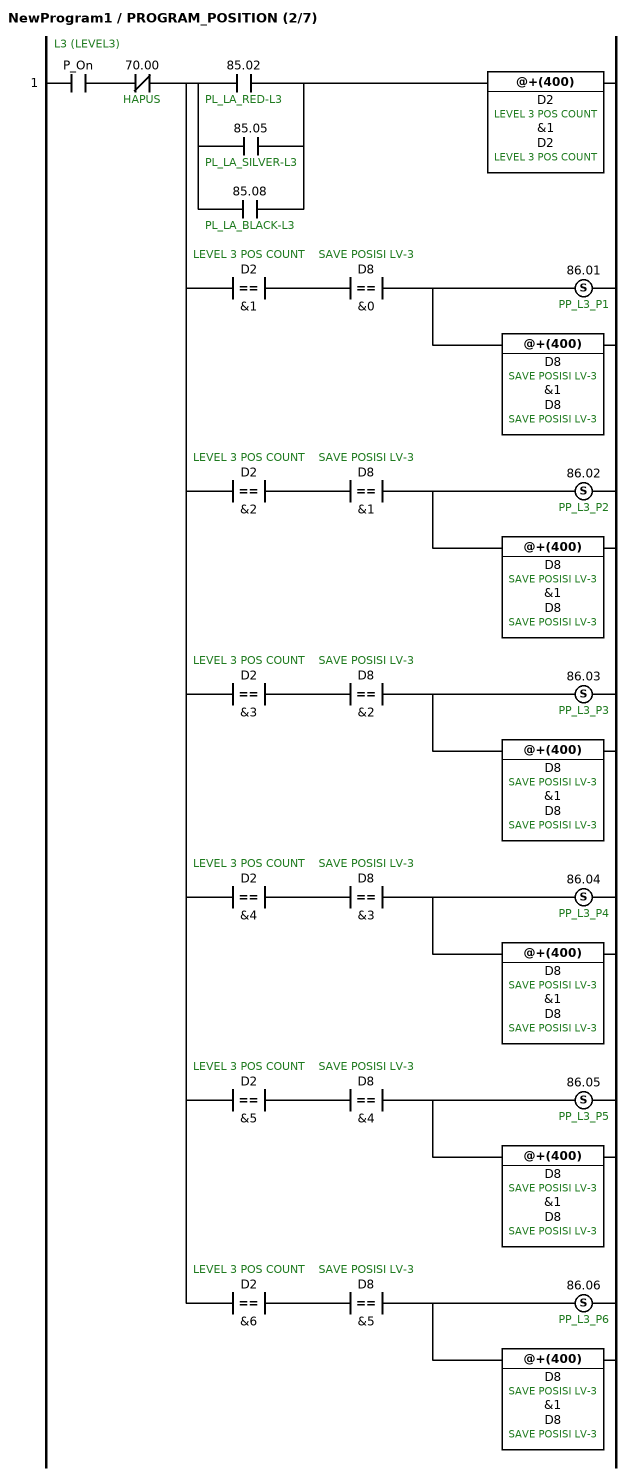
; rung 1: L3 (LEVEL3)
LD P_On
ANDNOT 70.00  ; HAPUS
OUT TR0
LD 85.02  ; PL_LA_RED-L3
OR 85.05  ; PL_LA_SILVER-L3
OR 85.08  ; PL_LA_BLACK-L3
ANDLD
@+(400) D2 &1 D2  ; LEVEL 3 POS COUNT
LD TR0
AND=(300) D2 &1  ; LEVEL 3 POS COUNT
AND=(300) D8 &0  ; SAVE POSISI LV-3
SET 86.01  ; PP_L3_P1
@+(400) D8 &1 D8  ; SAVE POSISI LV-3
LD TR0
AND=(300) D2 &2  ; LEVEL 3 POS COUNT
AND=(300) D8 &1  ; SAVE POSISI LV-3
SET 86.02  ; PP_L3_P2
@+(400) D8 &1 D8  ; SAVE POSISI LV-3
LD TR0
AND=(300) D2 &3  ; LEVEL 3 POS COUNT
AND=(300) D8 &2  ; SAVE POSISI LV-3
SET 86.03  ; PP_L3_P3
@+(400) D8 &1 D8  ; SAVE POSISI LV-3
LD TR0
AND=(300) D2 &4  ; LEVEL 3 POS COUNT
AND=(300) D8 &3  ; SAVE POSISI LV-3
SET 86.04  ; PP_L3_P4
@+(400) D8 &1 D8  ; SAVE POSISI LV-3
LD TR0
AND=(300) D2 &5  ; LEVEL 3 POS COUNT
AND=(300) D8 &4  ; SAVE POSISI LV-3
SET 86.05  ; PP_L3_P5
@+(400) D8 &1 D8  ; SAVE POSISI LV-3
LD TR0
AND=(300) D2 &6  ; LEVEL 3 POS COUNT
AND=(300) D8 &5  ; SAVE POSISI LV-3
SET 86.06  ; PP_L3_P6
@+(400) D8 &1 D8  ; SAVE POSISI LV-3

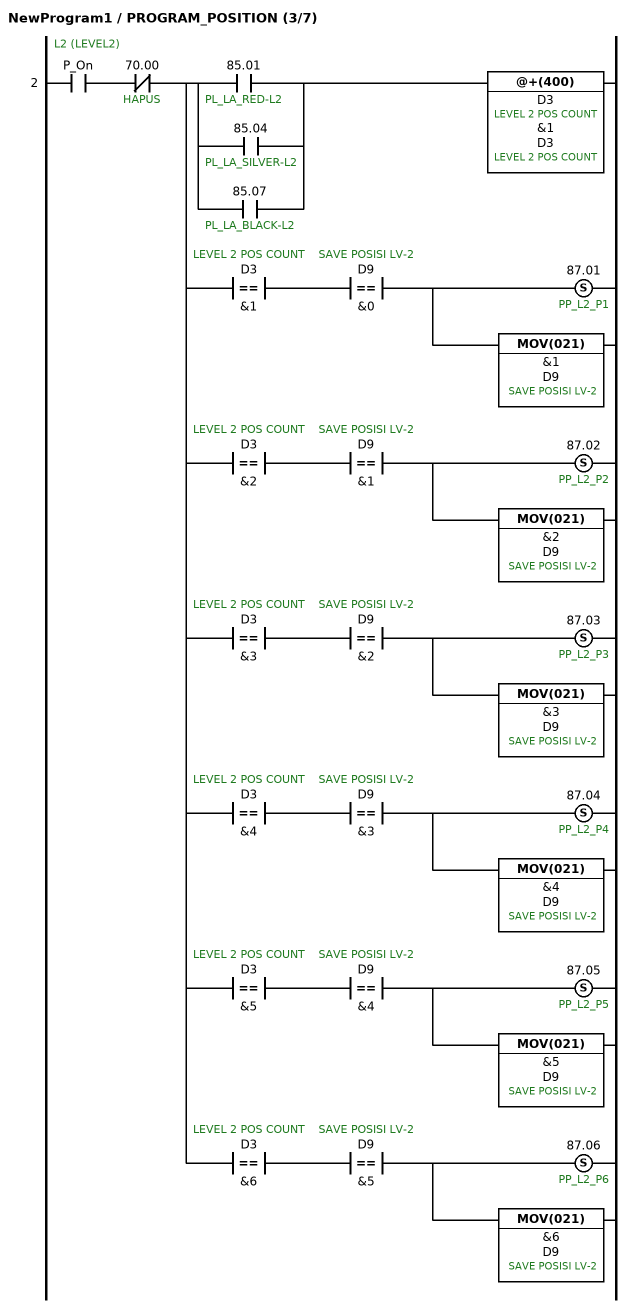
; rung 2: L2 (LEVEL2)
LD P_On
ANDNOT 70.00  ; HAPUS
OUT TR0
LD 85.01  ; PL_LA_RED-L2
OR 85.04  ; PL_LA_SILVER-L2
OR 85.07  ; PL_LA_BLACK-L2
ANDLD
@+(400) D3 &1 D3  ; LEVEL 2 POS COUNT
LD TR0
AND=(300) D3 &1  ; LEVEL 2 POS COUNT
AND=(300) D9 &0  ; SAVE POSISI LV-2
SET 87.01  ; PP_L2_P1
MOV(021) &1 D9  ; SAVE POSISI LV-2
LD TR0
AND=(300) D3 &2  ; LEVEL 2 POS COUNT
AND=(300) D9 &1  ; SAVE POSISI LV-2
SET 87.02  ; PP_L2_P2
MOV(021) &2 D9  ; SAVE POSISI LV-2
LD TR0
AND=(300) D3 &3  ; LEVEL 2 POS COUNT
AND=(300) D9 &2  ; SAVE POSISI LV-2
SET 87.03  ; PP_L2_P3
MOV(021) &3 D9  ; SAVE POSISI LV-2
LD TR0
AND=(300) D3 &4  ; LEVEL 2 POS COUNT
AND=(300) D9 &3  ; SAVE POSISI LV-2
SET 87.04  ; PP_L2_P4
MOV(021) &4 D9  ; SAVE POSISI LV-2
LD TR0
AND=(300) D3 &5  ; LEVEL 2 POS COUNT
AND=(300) D9 &4  ; SAVE POSISI LV-2
SET 87.05  ; PP_L2_P5
MOV(021) &5 D9  ; SAVE POSISI LV-2
LD TR0
AND=(300) D3 &6  ; LEVEL 2 POS COUNT
AND=(300) D9 &5  ; SAVE POSISI LV-2
SET 87.06  ; PP_L2_P6
MOV(021) &6 D9  ; SAVE POSISI LV-2

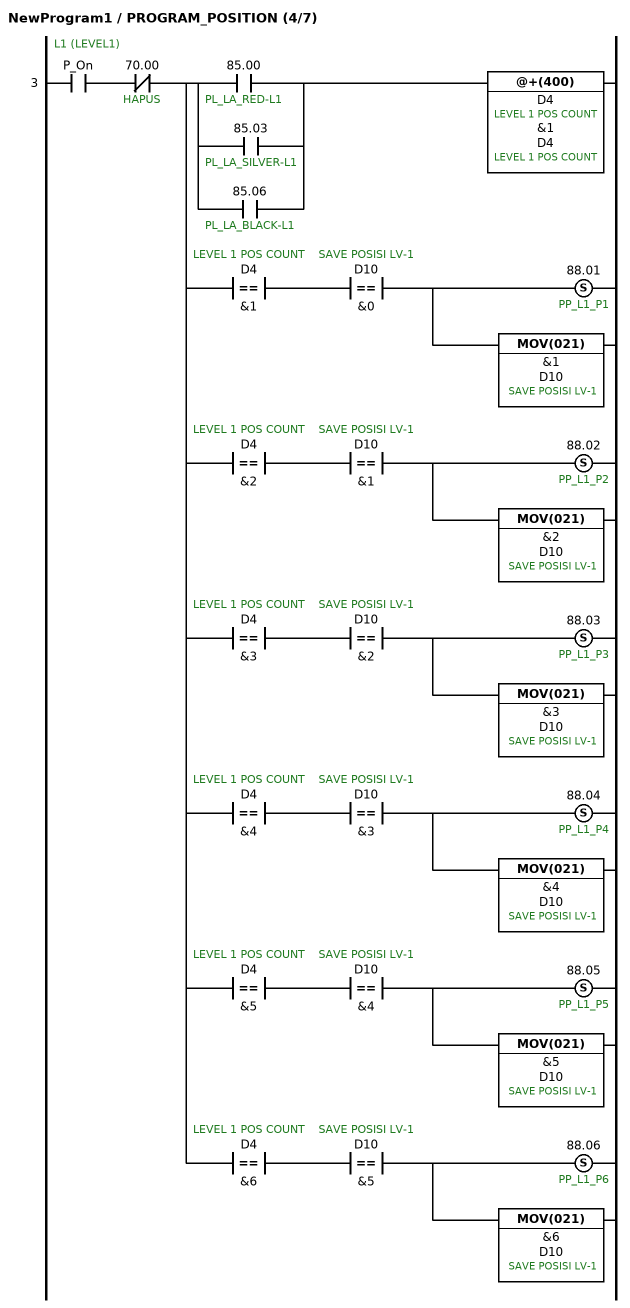
; rung 3: L1 (LEVEL1)
LD P_On
ANDNOT 70.00  ; HAPUS
OUT TR0
LD 85.00  ; PL_LA_RED-L1
OR 85.03  ; PL_LA_SILVER-L1
OR 85.06  ; PL_LA_BLACK-L1
ANDLD
@+(400) D4 &1 D4  ; LEVEL 1 POS COUNT
LD TR0
AND=(300) D4 &1  ; LEVEL 1 POS COUNT
AND=(300) D10 &0  ; SAVE POSISI LV-1
SET 88.01  ; PP_L1_P1
MOV(021) &1 D10  ; SAVE POSISI LV-1
LD TR0
AND=(300) D4 &2  ; LEVEL 1 POS COUNT
AND=(300) D10 &1  ; SAVE POSISI LV-1
SET 88.02  ; PP_L1_P2
MOV(021) &2 D10  ; SAVE POSISI LV-1
LD TR0
AND=(300) D4 &3  ; LEVEL 1 POS COUNT
AND=(300) D10 &2  ; SAVE POSISI LV-1
SET 88.03  ; PP_L1_P3
MOV(021) &3 D10  ; SAVE POSISI LV-1
LD TR0
AND=(300) D4 &4  ; LEVEL 1 POS COUNT
AND=(300) D10 &3  ; SAVE POSISI LV-1
SET 88.04  ; PP_L1_P4
MOV(021) &4 D10  ; SAVE POSISI LV-1
LD TR0
AND=(300) D4 &5  ; LEVEL 1 POS COUNT
AND=(300) D10 &4  ; SAVE POSISI LV-1
SET 88.05  ; PP_L1_P5
MOV(021) &5 D10  ; SAVE POSISI LV-1
LD TR0
AND=(300) D4 &6  ; LEVEL 1 POS COUNT
AND=(300) D10 &5  ; SAVE POSISI LV-1
SET 88.06  ; PP_L1_P6
MOV(021) &6 D10  ; SAVE POSISI LV-1

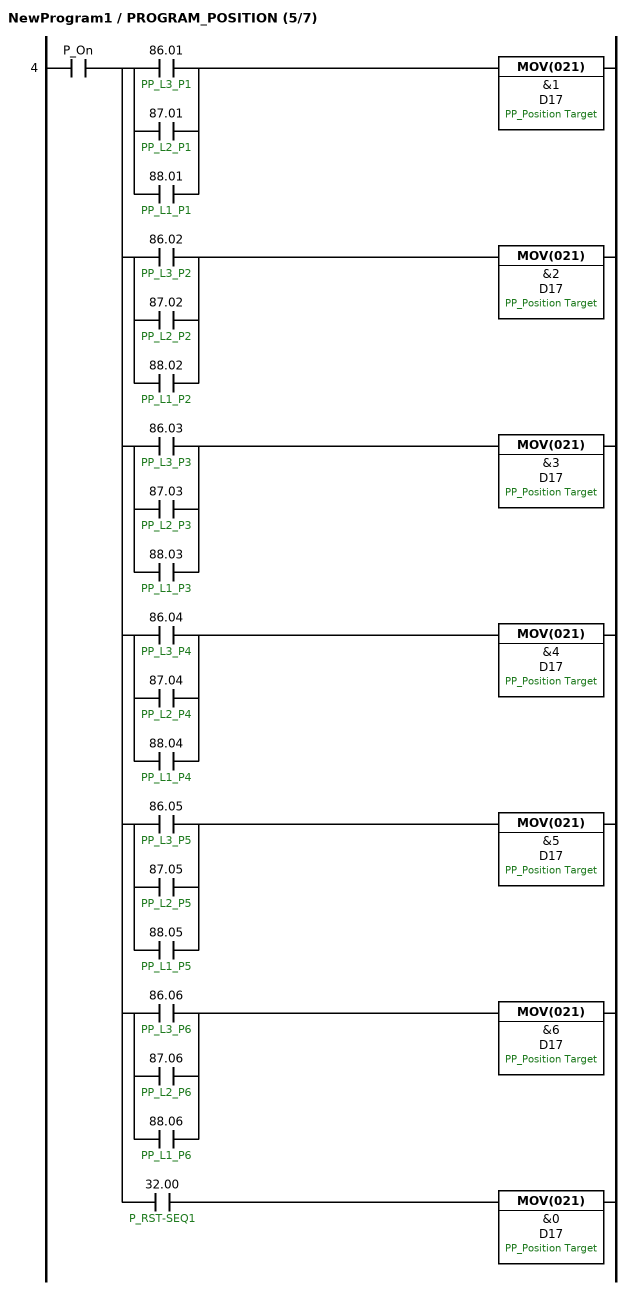
; rung 4
LD P_On
OUT TR0
LD 86.01  ; PP_L3_P1
OR 87.01  ; PP_L2_P1
OR 88.01  ; PP_L1_P1
ANDLD
MOV(021) &1 D17  ; PP_Position Target
LD TR0
LD 86.02  ; PP_L3_P2
OR 87.02  ; PP_L2_P2
OR 88.02  ; PP_L1_P2
ANDLD
MOV(021) &2 D17  ; PP_Position Target
LD TR0
LD 86.03  ; PP_L3_P3
OR 87.03  ; PP_L2_P3
OR 88.03  ; PP_L1_P3
ANDLD
MOV(021) &3 D17  ; PP_Position Target
LD TR0
LD 86.04  ; PP_L3_P4
OR 87.04  ; PP_L2_P4
OR 88.04  ; PP_L1_P4
ANDLD
MOV(021) &4 D17  ; PP_Position Target
LD TR0
LD 86.05  ; PP_L3_P5
OR 87.05  ; PP_L2_P5
OR 88.05  ; PP_L1_P5
ANDLD
MOV(021) &5 D17  ; PP_Position Target
LD TR0
LD 86.06  ; PP_L3_P6
OR 87.06  ; PP_L2_P6
OR 88.06  ; PP_L1_P6
ANDLD
MOV(021) &6 D17  ; PP_Position Target
LD TR0
AND 32.00  ; P_RST-SEQ1
MOV(021) &0 D17  ; PP_Position Target

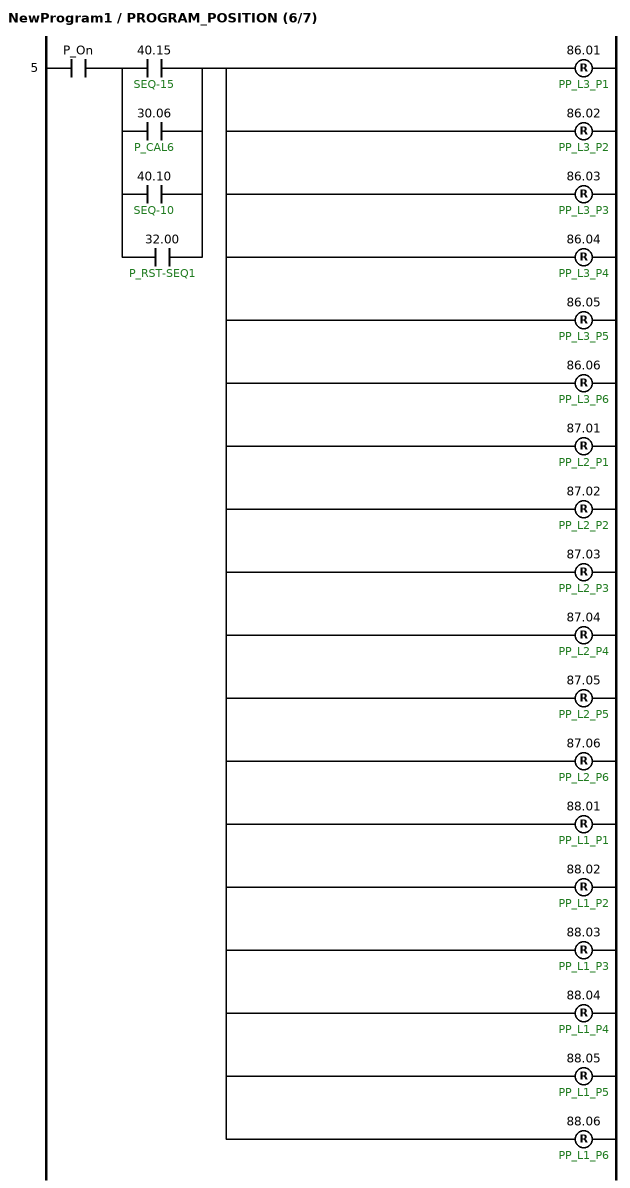
; rung 5
LD P_On
LD 40.15  ; SEQ-15
OR 30.06  ; P_CAL6
OR 40.10  ; SEQ-10
OR 32.00  ; P_RST-SEQ1
ANDLD
RSET 86.01  ; PP_L3_P1
RSET 86.02  ; PP_L3_P2
RSET 86.03  ; PP_L3_P3
RSET 86.04  ; PP_L3_P4
RSET 86.05  ; PP_L3_P5
RSET 86.06  ; PP_L3_P6
RSET 87.01  ; PP_L2_P1
RSET 87.02  ; PP_L2_P2
RSET 87.03  ; PP_L2_P3
RSET 87.04  ; PP_L2_P4
RSET 87.05  ; PP_L2_P5
RSET 87.06  ; PP_L2_P6
RSET 88.01  ; PP_L1_P1
RSET 88.02  ; PP_L1_P2
RSET 88.03  ; PP_L1_P3
RSET 88.04  ; PP_L1_P4
RSET 88.05  ; PP_L1_P5
RSET 88.06  ; PP_L1_P6

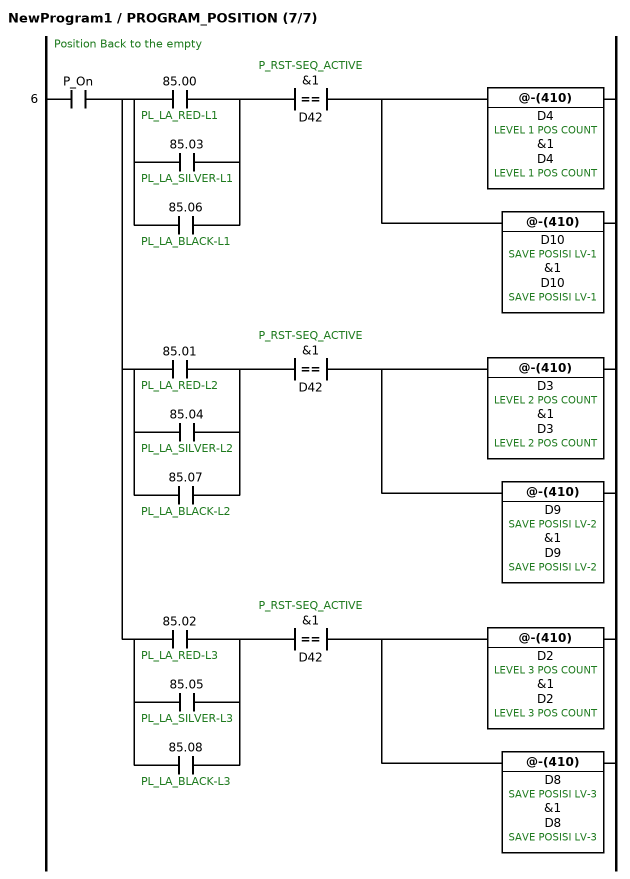
; rung 6: Position Back to the empty
LD P_On
OUT TR0
LD 85.00  ; PL_LA_RED-L1
OR 85.03  ; PL_LA_SILVER-L1
OR 85.06  ; PL_LA_BLACK-L1
ANDLD
AND=(300) &1 D42  ; P_RST-SEQ_ACTIVE
@-(410) D4 &1 D4  ; LEVEL 1 POS COUNT
@-(410) D10 &1 D10  ; SAVE POSISI LV-1
LD TR0
LD 85.01  ; PL_LA_RED-L2
OR 85.04  ; PL_LA_SILVER-L2
OR 85.07  ; PL_LA_BLACK-L2
ANDLD
AND=(300) &1 D42  ; P_RST-SEQ_ACTIVE
@-(410) D3 &1 D3  ; LEVEL 2 POS COUNT
@-(410) D9 &1 D9  ; SAVE POSISI LV-2
LD TR0
LD 85.02  ; PL_LA_RED-L3
OR 85.05  ; PL_LA_SILVER-L3
OR 85.08  ; PL_LA_BLACK-L3
ANDLD
AND=(300) &1 D42  ; P_RST-SEQ_ACTIVE
@-(410) D2 &1 D2  ; LEVEL 3 POS COUNT
@-(410) D8 &1 D8  ; SAVE POSISI LV-3

### Section SEQ_HORIZONTAL

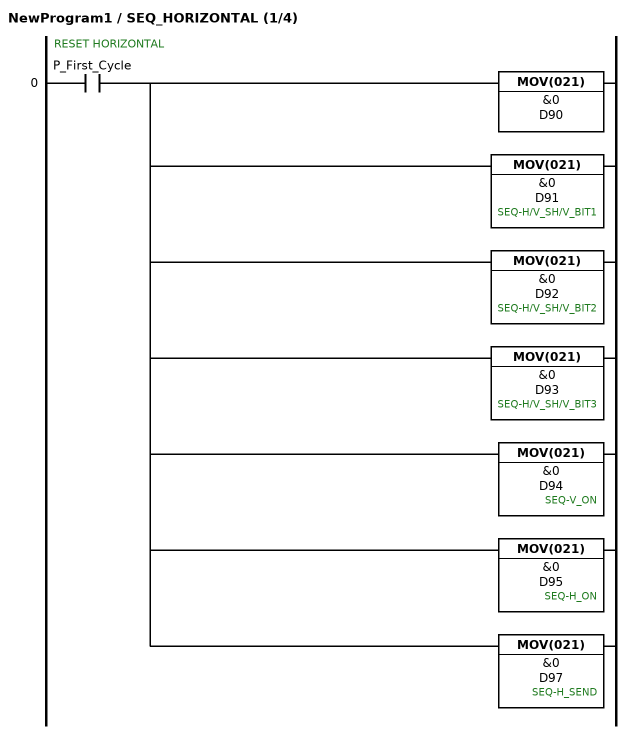
; rung 0: RESET HORIZONTAL
LD P_First_Cycle
MOV(021) &0 D90
MOV(021) &0 D91  ; SEQ-H/V_SH/V_BIT1
MOV(021) &0 D92  ; SEQ-H/V_SH/V_BIT2
MOV(021) &0 D93  ; SEQ-H/V_SH/V_BIT3
MOV(021) &0 D94  ; SEQ-V_ON
MOV(021) &0 D95  ; SEQ-H_ON
MOV(021) &0 D97  ; SEQ-H_SEND

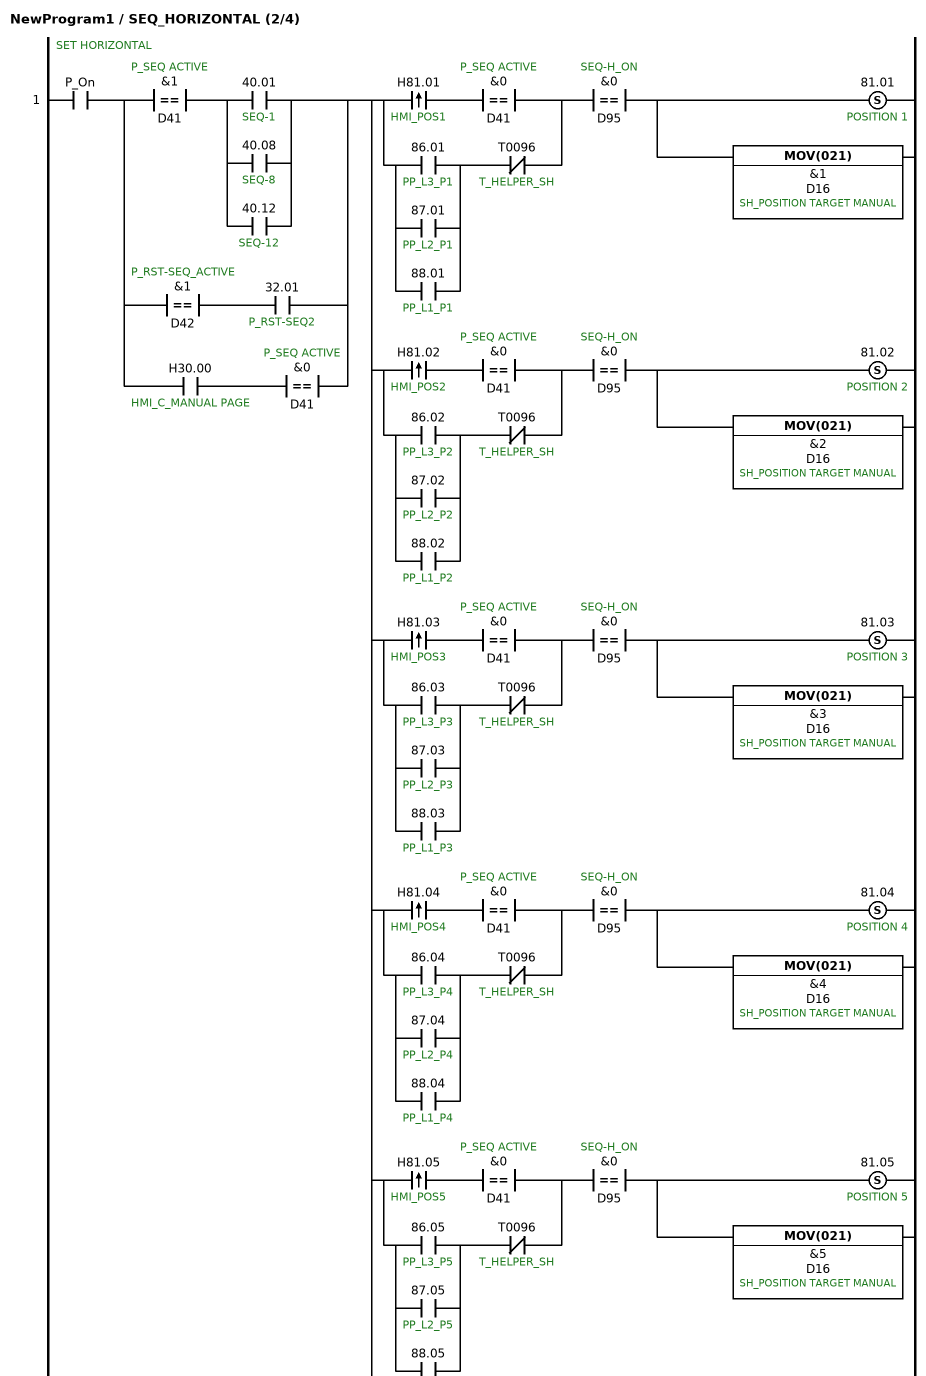

